   1:  PR[GP1:91,1] = PR[GP1:90,1] + -28.583;
   1:  PR[GP1:91,2] = PR[GP1:90,2] + 39.031;
   1:L PR[91] 10mm/sec CNT100;
   1:  PR[GP1:91,1] = PR[GP1:90,1] + -29.750;
   1:  PR[GP1:91,2] = PR[GP1:90,2] + 38.604;
   1:L PR[91] 10mm/sec CNT100;
   1:  PR[GP1:91,1] = PR[GP1:90,1] + -40.400;
   1:  PR[GP1:91,2] = PR[GP1:90,2] + 33.947;
   1:L PR[91] 10mm/sec CNT100;
   1:  PR[GP1:91,1] = PR[GP1:90,1] + -41.704;
   1:  PR[GP1:91,2] = PR[GP1:90,2] + 33.125;
   1:L PR[91] 10mm/sec CNT100;
   1:  PR[GP1:91,1] = PR[GP1:90,1] + -42.919;
   1:  PR[GP1:91,2] = PR[GP1:90,2] + 31.940;
   1:L PR[91] 10mm/sec CNT100;
   1:  PR[GP1:91,1] = PR[GP1:90,1] + -51.021;
   1:  PR[GP1:91,2] = PR[GP1:90,2] + 24.604;
   1:L PR[91] 10mm/sec CNT100;
   1:  PR[GP1:91,1] = PR[GP1:90,1] + -52.053;
   1:  PR[GP1:91,2] = PR[GP1:90,2] + 22.993;
   1:L PR[91] 10mm/sec CNT100;
   1:  PR[GP1:91,1] = PR[GP1:90,1] + -57.032;
   1:  PR[GP1:91,2] = PR[GP1:90,2] + 13.999;
   1:L PR[91] 10mm/sec CNT100;
   1:  PR[GP1:91,1] = PR[GP1:90,1] + -57.722;
   1:  PR[GP1:91,2] = PR[GP1:90,2] + 12.097;
   1:L PR[91] 10mm/sec CNT100;
   1:  PR[GP1:91,1] = PR[GP1:90,1] + -57.950;
   1:  PR[GP1:91,2] = PR[GP1:90,2] + 10.064;
   1:L PR[91] 10mm/sec CNT100;
   1:  PR[GP1:91,1] = PR[GP1:90,1] + -59.627;
   1:  PR[GP1:91,2] = PR[GP1:90,2] + 0.261;
   1:L PR[91] 10mm/sec CNT100;
   1:  PR[GP1:91,1] = PR[GP1:90,1] + -59.403;
   1:  PR[GP1:91,2] = PR[GP1:90,2] + -1.752;
   1:L PR[91] 10mm/sec CNT100;
   1:  PR[GP1:91,1] = PR[GP1:90,1] + -57.736;
   1:  PR[GP1:91,2] = PR[GP1:90,2] + -11.502;
   1:L PR[91] 10mm/sec CNT100;
   1:  PR[GP1:91,1] = PR[GP1:90,1] + -57.039;
   1:  PR[GP1:91,2] = PR[GP1:90,2] + -13.421;
   1:L PR[91] 10mm/sec CNT100;
   1:  PR[GP1:91,1] = PR[GP1:90,1] + -52.081;
   1:  PR[GP1:91,2] = PR[GP1:90,2] + -22.399;
   1:L PR[91] 10mm/sec CNT100;
   1:  PR[GP1:91,1] = PR[GP1:90,1] + -51.042;
   1:  PR[GP1:91,2] = PR[GP1:90,2] + -24.020;
   1:L PR[91] 10mm/sec CNT100;
   1:  PR[GP1:91,1] = PR[GP1:90,1] + -49.777;
   1:  PR[GP1:91,2] = PR[GP1:90,2] + -25.262;
   1:L PR[91] 10mm/sec CNT100;
   1:  PR[GP1:91,1] = PR[GP1:90,1] + -41.775;
   1:  PR[GP1:91,2] = PR[GP1:90,2] + -32.521;
   1:L PR[91] 10mm/sec CNT100;
   1:  PR[GP1:91,1] = PR[GP1:90,1] + -40.461;
   1:  PR[GP1:91,2] = PR[GP1:90,2] + -33.350;
   1:L PR[91] 10mm/sec CNT100;
   1:  PR[GP1:91,1] = PR[GP1:90,1] + -29.851;
   1:  PR[GP1:91,2] = PR[GP1:90,2] + -38.019;
   1:L PR[91] 10mm/sec CNT100;
   1:  PR[GP1:91,1] = PR[GP1:90,1] + -28.670;
   1:  PR[GP1:91,2] = PR[GP1:90,2] + -38.452;
   1:L PR[91] 10mm/sec CNT100;
   1:  PR[GP1:91,1] = PR[GP1:90,1] + -27.548;
   1:  PR[GP1:91,2] = PR[GP1:90,2] + -38.612;
   1:L PR[91] 10mm/sec CNT100;
   1:  PR[GP1:91,1] = PR[GP1:90,1] + -15.395;
   1:  PR[GP1:91,2] = PR[GP1:90,2] + -39.778;
   1:L PR[91] 10mm/sec CNT100;
   1:  PR[GP1:91,1] = PR[GP1:90,1] + -14.616;
   1:  PR[GP1:91,2] = PR[GP1:90,2] + -39.726;
   1:L PR[91] 10mm/sec CNT100;
   1:  PR[GP1:91,1] = PR[GP1:90,1] + -2.012;
   1:  PR[GP1:91,2] = PR[GP1:90,2] + -36.843;
   1:L PR[91] 10mm/sec CNT100;
   1:  PR[GP1:91,1] = PR[GP1:90,1] + -1.587;
   1:  PR[GP1:91,2] = PR[GP1:90,2] + -36.721;
   1:L PR[91] 10mm/sec CNT100;
   1:  PR[GP1:91,1] = PR[GP1:90,1] + -0.264;
   1:  PR[GP1:91,2] = PR[GP1:90,2] + -35.946;
   1:L PR[91] 10mm/sec CNT100;
   1:  PR[GP1:91,1] = PR[GP1:90,1] + 0.805;
   1:  PR[GP1:91,2] = PR[GP1:90,2] + -36.790;
   1:  PR[GP1:91,3] = PR[GP1:90,3] + 82.655;
   1:L PR[91] 10mm/sec CNT100;
   1:  PR[GP1:91,1] = PR[GP1:90,1] + 1.110;
   1:  PR[GP1:91,2] = PR[GP1:90,2] + -36.877;
   1:L PR[91] 10mm/sec CNT100;
   1:  PR[GP1:91,1] = PR[GP1:90,1] + 13.913;
   1:  PR[GP1:91,2] = PR[GP1:90,2] + -39.807;
   1:L PR[91] 10mm/sec CNT100;
   1:  PR[GP1:91,1] = PR[GP1:90,1] + 14.554;
   1:  PR[GP1:91,2] = PR[GP1:90,2] + -39.849;
   1:L PR[91] 10mm/sec CNT100;
   1:  PR[GP1:91,1] = PR[GP1:90,1] + 15.335;
   1:  PR[GP1:91,2] = PR[GP1:90,2] + -39.742;
   1:L PR[91] 10mm/sec CNT100;
   1:  PR[GP1:91,1] = PR[GP1:90,1] + 27.932;
   1:  PR[GP1:91,2] = PR[GP1:90,2] + -38.517;
   1:L PR[91] 10mm/sec CNT100;
   1:  PR[GP1:91,1] = PR[GP1:90,1] + 28.976;
   1:  PR[GP1:91,2] = PR[GP1:90,2] + -38.137;
   1:L PR[91] 10mm/sec CNT100;
   1:  PR[GP1:91,1] = PR[GP1:90,1] + 39.784;
   1:  PR[GP1:91,2] = PR[GP1:90,2] + -33.383;
   1:L PR[91] 10mm/sec CNT100;
   1:  PR[GP1:91,1] = PR[GP1:90,1] + 40.970;
   1:  PR[GP1:91,2] = PR[GP1:90,2] + -32.639;
   1:L PR[91] 10mm/sec CNT100;
   1:  PR[GP1:91,1] = PR[GP1:90,1] + 42.083;
   1:  PR[GP1:91,2] = PR[GP1:90,2] + -31.555;
   1:L PR[91] 10mm/sec CNT100;
   1:  PR[GP1:91,1] = PR[GP1:90,1] + 50.319;
   1:  PR[GP1:91,2] = PR[GP1:90,2] + -24.063;
   1:L PR[91] 10mm/sec CNT100;
   1:  PR[GP1:91,1] = PR[GP1:90,1] + 51.288;
   1:  PR[GP1:91,2] = PR[GP1:90,2] + -22.560;
   1:L PR[91] 10mm/sec CNT100;
   1:  PR[GP1:91,1] = PR[GP1:90,1] + 56.354;
   1:  PR[GP1:91,2] = PR[GP1:90,2] + -13.404;
   1:L PR[91] 10mm/sec CNT100;
   1:  PR[GP1:91,1] = PR[GP1:90,1] + 56.995;
   1:  PR[GP1:91,2] = PR[GP1:90,2] + -11.659;
   1:L PR[91] 10mm/sec CNT100;
   1:  PR[GP1:91,1] = PR[GP1:90,1] + 57.216;
   1:  PR[GP1:91,2] = PR[GP1:90,2] + -9.715;
   1:L PR[91] 10mm/sec CNT100;
   1:  PR[GP1:91,1] = PR[GP1:90,1] + 58.924;
   1:  PR[GP1:91,2] = PR[GP1:90,2] + 0.296;
   1:L PR[91] 10mm/sec CNT100;
   1:  PR[GP1:91,1] = PR[GP1:90,1] + 58.706;
   1:  PR[GP1:91,2] = PR[GP1:90,2] + 2.224;
   1:L PR[91] 10mm/sec CNT100;
   1:  PR[GP1:91,1] = PR[GP1:90,1] + 56.994;
   1:  PR[GP1:91,2] = PR[GP1:90,2] + 12.222;
   1:L PR[91] 10mm/sec CNT100;
   1:  PR[GP1:91,1] = PR[GP1:90,1] + 56.346;
   1:  PR[GP1:91,2] = PR[GP1:90,2] + 13.982;
   1:L PR[91] 10mm/sec CNT100;
   1:  PR[GP1:91,1] = PR[GP1:90,1] + 51.259;
   1:  PR[GP1:91,2] = PR[GP1:90,2] + 23.154;
   1:L PR[91] 10mm/sec CNT100;
   1:  PR[GP1:91,1] = PR[GP1:90,1] + 50.284;
   1:  PR[GP1:91,2] = PR[GP1:90,2] + 24.667;
   1:L PR[91] 10mm/sec CNT100;
   1:  PR[GP1:91,1] = PR[GP1:90,1] + 49.110;
   1:  PR[GP1:91,2] = PR[GP1:90,2] + 25.817;
   1:L PR[91] 10mm/sec CNT100;
   1:  PR[GP1:91,1] = PR[GP1:90,1] + 40.917;
   1:  PR[GP1:91,2] = PR[GP1:90,2] + 33.232;
   1:L PR[91] 10mm/sec CNT100;
   1:  PR[GP1:91,1] = PR[GP1:90,1] + 39.723;
   1:  PR[GP1:91,2] = PR[GP1:90,2] + 33.981;
   1:L PR[91] 10mm/sec CNT100;
   1:  PR[GP1:91,1] = PR[GP1:90,1] + 28.873;
   1:  PR[GP1:91,2] = PR[GP1:90,2] + 38.722;
   1:L PR[91] 10mm/sec CNT100;
   1:  PR[GP1:91,1] = PR[GP1:90,1] + 27.818;
   1:  PR[GP1:91,2] = PR[GP1:90,2] + 39.107;
   1:L PR[91] 10mm/sec CNT100;
   1:  PR[GP1:91,1] = PR[GP1:90,1] + 26.822;
   1:  PR[GP1:91,2] = PR[GP1:90,2] + 39.248;
   1:L PR[91] 10mm/sec CNT100;
   1:  PR[GP1:91,1] = PR[GP1:90,1] + 14.428;
   1:  PR[GP1:91,2] = PR[GP1:90,2] + 40.400;
   1:L PR[91] 10mm/sec CNT100;
   1:  PR[GP1:91,1] = PR[GP1:90,1] + 13.778;
   1:  PR[GP1:91,2] = PR[GP1:90,2] + 40.356;
   1:L PR[91] 10mm/sec CNT100;
   1:  PR[GP1:91,1] = PR[GP1:90,1] + 0.766;
   1:  PR[GP1:91,2] = PR[GP1:90,2] + 37.283;
   1:L PR[91] 10mm/sec CNT100;
   1:  PR[GP1:91,1] = PR[GP1:90,1] + 0.557;
   1:  PR[GP1:91,2] = PR[GP1:90,2] + 37.223;
   1:L PR[91] 10mm/sec CNT100;
   1:  PR[GP1:91,1] = PR[GP1:90,1] + -0.262;
   1:  PR[GP1:91,2] = PR[GP1:90,2] + 36.794;
   1:L PR[91] 10mm/sec CNT100;
   1:  PR[GP1:91,1] = PR[GP1:90,1] + -1.079;
   1:  PR[GP1:91,2] = PR[GP1:90,2] + 37.223;
   1:L PR[91] 10mm/sec CNT100;
   1:  PR[GP1:91,1] = PR[GP1:90,1] + -1.288;
   1:  PR[GP1:91,2] = PR[GP1:90,2] + 37.283;
   1:L PR[91] 10mm/sec CNT100;
   1:  PR[GP1:91,1] = PR[GP1:90,1] + -14.303;
   1:  PR[GP1:91,2] = PR[GP1:90,2] + 40.356;
   1:L PR[91] 10mm/sec CNT100;
   1:  PR[GP1:91,1] = PR[GP1:90,1] + -14.942;
   1:  PR[GP1:91,2] = PR[GP1:90,2] + 40.398;
   1:L PR[91] 10mm/sec CNT100;
   1:  PR[GP1:91,1] = PR[GP1:90,1] + -15.723;
   1:  PR[GP1:91,2] = PR[GP1:90,2] + 40.290;
   1:L PR[91] 10mm/sec CNT100;
   1:  PR[GP1:91,1] = PR[GP1:90,1] + -28.363;
   1:  PR[GP1:91,2] = PR[GP1:90,2] + 39.102;
   1:L PR[91] 10mm/sec CNT100;
   1:  PR[GP1:91,1] = PR[GP1:90,1] + -29.403;
   1:  PR[GP1:91,2] = PR[GP1:90,2] + 38.721;
   1:L PR[91] 10mm/sec CNT100;
   1:  PR[GP1:91,1] = PR[GP1:90,1] + -40.254;
   1:  PR[GP1:91,2] = PR[GP1:90,2] + 33.977;
   1:L PR[91] 10mm/sec CNT100;
   1:  PR[GP1:91,1] = PR[GP1:90,1] + -41.446;
   1:  PR[GP1:91,2] = PR[GP1:90,2] + 33.225;
   1:L PR[91] 10mm/sec CNT100;
   1:  PR[GP1:91,1] = PR[GP1:90,1] + -42.561;
   1:  PR[GP1:91,2] = PR[GP1:90,2] + 32.136;
   1:L PR[91] 10mm/sec CNT100;
   1:  PR[GP1:91,1] = PR[GP1:90,1] + -50.832;
   1:  PR[GP1:91,2] = PR[GP1:90,2] + 24.648;
   1:L PR[91] 10mm/sec CNT100;
   1:  PR[GP1:91,1] = PR[GP1:90,1] + -51.790;
   1:  PR[GP1:91,2] = PR[GP1:90,2] + 23.152;
   1:L PR[91] 10mm/sec CNT100;
   1:  PR[GP1:91,1] = PR[GP1:90,1] + -56.877;
   1:  PR[GP1:91,2] = PR[GP1:90,2] + 13.963;
   1:L PR[91] 10mm/sec CNT100;
   1:  PR[GP1:91,1] = PR[GP1:90,1] + -57.522;
   1:  PR[GP1:91,2] = PR[GP1:90,2] + 12.187;
   1:L PR[91] 10mm/sec CNT100;
   1:  PR[GP1:91,1] = PR[GP1:90,1] + -57.735;
   1:  PR[GP1:91,2] = PR[GP1:90,2] + 10.284;
   1:L PR[91] 10mm/sec CNT100;
   1:  PR[GP1:91,1] = PR[GP1:90,1] + -59.450;
   1:  PR[GP1:91,2] = PR[GP1:90,2] + 0.261;
   1:L PR[91] 10mm/sec CNT100;
   1:  PR[GP1:91,1] = PR[GP1:90,1] + -59.240;
   1:  PR[GP1:91,2] = PR[GP1:90,2] + -1.624;
   1:L PR[91] 10mm/sec CNT100;
   1:  PR[GP1:91,1] = PR[GP1:90,1] + -57.535;
   1:  PR[GP1:91,2] = PR[GP1:90,2] + -11.591;
   1:L PR[91] 10mm/sec CNT100;
   1:  PR[GP1:91,1] = PR[GP1:90,1] + -56.885;
   1:  PR[GP1:91,2] = PR[GP1:90,2] + -13.384;
   1:L PR[91] 10mm/sec CNT100;
   1:  PR[GP1:91,1] = PR[GP1:90,1] + -51.819;
   1:  PR[GP1:91,2] = PR[GP1:90,2] + -22.557;
   1:L PR[91] 10mm/sec CNT100;
   1:  PR[GP1:91,1] = PR[GP1:90,1] + -50.854;
   1:  PR[GP1:91,2] = PR[GP1:90,2] + -24.063;
   1:L PR[91] 10mm/sec CNT100;
   1:  PR[GP1:91,1] = PR[GP1:90,1] + -49.679;
   1:  PR[GP1:91,2] = PR[GP1:90,2] + -25.217;
   1:L PR[91] 10mm/sec CNT100;
   1:  PR[GP1:91,1] = PR[GP1:90,1] + -41.518;
   1:  PR[GP1:91,2] = PR[GP1:90,2] + -32.620;
   1:L PR[91] 10mm/sec CNT100;
   1:  PR[GP1:91,1] = PR[GP1:90,1] + -40.315;
   1:  PR[GP1:91,2] = PR[GP1:90,2] + -33.379;
   1:L PR[91] 10mm/sec CNT100;
   1:  PR[GP1:91,1] = PR[GP1:90,1] + -29.506;
   1:  PR[GP1:91,2] = PR[GP1:90,2] + -38.135;
   1:L PR[91] 10mm/sec CNT100;
   1:  PR[GP1:91,1] = PR[GP1:90,1] + -28.451;
   1:  PR[GP1:91,2] = PR[GP1:90,2] + -38.522;
   1:L PR[91] 10mm/sec CNT100;
   1:  PR[GP1:91,1] = PR[GP1:90,1] + -27.450;
   1:  PR[GP1:91,2] = PR[GP1:90,2] + -38.664;
   1:L PR[91] 10mm/sec CNT100;
   1:  PR[GP1:91,1] = PR[GP1:90,1] + -15.095;
   1:  PR[GP1:91,2] = PR[GP1:90,2] + -39.850;
   1:L PR[91] 10mm/sec CNT100;
   1:  PR[GP1:91,1] = PR[GP1:90,1] + -14.439;
   1:  PR[GP1:91,2] = PR[GP1:90,2] + -39.806;
   1:L PR[91] 10mm/sec CNT100;
   1:  PR[GP1:91,1] = PR[GP1:90,1] + -1.637;
   1:  PR[GP1:91,2] = PR[GP1:90,2] + -36.877;
   1:L PR[91] 10mm/sec CNT100;
   1:  PR[GP1:91,1] = PR[GP1:90,1] + -1.332;
   1:  PR[GP1:91,2] = PR[GP1:90,2] + -36.790;
   1:L PR[91] 10mm/sec CNT100;
   1:  PR[GP1:91,1] = PR[GP1:90,1] + -0.264;
   1:  PR[GP1:91,2] = PR[GP1:90,2] + -36.164;
   1:L PR[91] 10mm/sec CNT100;
   1:  PR[GP1:91,1] = PR[GP1:90,1] + 0.550;
   1:  PR[GP1:91,2] = PR[GP1:90,2] + -36.859;
   1:  PR[GP1:91,3] = PR[GP1:90,3] + 83.265;
   1:L PR[91] 10mm/sec CNT100;
   1:  PR[GP1:91,1] = PR[GP1:90,1] + 0.735;
   1:  PR[GP1:91,2] = PR[GP1:90,2] + -36.912;
   1:L PR[91] 10mm/sec CNT100;
   1:  PR[GP1:91,1] = PR[GP1:90,1] + 13.736;
   1:  PR[GP1:91,2] = PR[GP1:90,2] + -39.887;
   1:L PR[91] 10mm/sec CNT100;
   1:  PR[GP1:91,1] = PR[GP1:90,1] + 14.254;
   1:  PR[GP1:91,2] = PR[GP1:90,2] + -39.921;
   1:L PR[91] 10mm/sec CNT100;
   1:  PR[GP1:91,1] = PR[GP1:90,1] + 14.899;
   1:  PR[GP1:91,2] = PR[GP1:90,2] + -39.832;
   1:L PR[91] 10mm/sec CNT100;
   1:  PR[GP1:91,1] = PR[GP1:90,1] + 27.715;
   1:  PR[GP1:91,2] = PR[GP1:90,2] + -38.587;
   1:L PR[91] 10mm/sec CNT100;
   1:  PR[GP1:91,1] = PR[GP1:90,1] + 28.632;
   1:  PR[GP1:91,2] = PR[GP1:90,2] + -38.252;
   1:L PR[91] 10mm/sec CNT100;
   1:  PR[GP1:91,1] = PR[GP1:90,1] + 39.639;
   1:  PR[GP1:91,2] = PR[GP1:90,2] + -33.412;
   1:L PR[91] 10mm/sec CNT100;
   1:  PR[GP1:91,1] = PR[GP1:90,1] + 40.715;
   1:  PR[GP1:91,2] = PR[GP1:90,2] + -32.737;
   1:L PR[91] 10mm/sec CNT100;
   1:  PR[GP1:91,1] = PR[GP1:90,1] + 41.728;
   1:  PR[GP1:91,2] = PR[GP1:90,2] + -31.749;
   1:L PR[91] 10mm/sec CNT100;
   1:  PR[GP1:91,1] = PR[GP1:90,1] + 50.132;
   1:  PR[GP1:91,2] = PR[GP1:90,2] + -24.105;
   1:L PR[91] 10mm/sec CNT100;
   1:  PR[GP1:91,1] = PR[GP1:90,1] + 51.027;
   1:  PR[GP1:91,2] = PR[GP1:90,2] + -22.717;
   1:L PR[91] 10mm/sec CNT100;
   1:  PR[GP1:91,1] = PR[GP1:90,1] + 56.200;
   1:  PR[GP1:91,2] = PR[GP1:90,2] + -13.367;
   1:L PR[91] 10mm/sec CNT100;
   1:  PR[GP1:91,1] = PR[GP1:90,1] + 56.796;
   1:  PR[GP1:91,2] = PR[GP1:90,2] + -11.746;
   1:L PR[91] 10mm/sec CNT100;
   1:  PR[GP1:91,1] = PR[GP1:90,1] + 57.002;
   1:  PR[GP1:91,2] = PR[GP1:90,2] + -9.935;
   1:L PR[91] 10mm/sec CNT100;
   1:  PR[GP1:91,1] = PR[GP1:90,1] + 58.747;
   1:  PR[GP1:91,2] = PR[GP1:90,2] + 0.296;
   1:L PR[91] 10mm/sec CNT100;
   1:  PR[GP1:91,1] = PR[GP1:90,1] + 58.543;
   1:  PR[GP1:91,2] = PR[GP1:90,2] + 2.093;
   1:L PR[91] 10mm/sec CNT100;
   1:  PR[GP1:91,1] = PR[GP1:90,1] + 56.794;
   1:  PR[GP1:91,2] = PR[GP1:90,2] + 12.309;
   1:L PR[91] 10mm/sec CNT100;
   1:  PR[GP1:91,1] = PR[GP1:90,1] + 56.192;
   1:  PR[GP1:91,2] = PR[GP1:90,2] + 13.946;
   1:L PR[91] 10mm/sec CNT100;
   1:  PR[GP1:91,1] = PR[GP1:90,1] + 50.997;
   1:  PR[GP1:91,2] = PR[GP1:90,2] + 23.313;
   1:L PR[91] 10mm/sec CNT100;
   1:  PR[GP1:91,1] = PR[GP1:90,1] + 50.096;
   1:  PR[GP1:91,2] = PR[GP1:90,2] + 24.710;
   1:L PR[91] 10mm/sec CNT100;
   1:  PR[GP1:91,1] = PR[GP1:90,1] + 49.013;
   1:  PR[GP1:91,2] = PR[GP1:90,2] + 25.771;
   1:L PR[91] 10mm/sec CNT100;
   1:  PR[GP1:91,1] = PR[GP1:90,1] + 40.660;
   1:  PR[GP1:91,2] = PR[GP1:90,2] + 33.330;
   1:L PR[91] 10mm/sec CNT100;
   1:  PR[GP1:91,1] = PR[GP1:90,1] + 39.577;
   1:  PR[GP1:91,2] = PR[GP1:90,2] + 34.010;
   1:L PR[91] 10mm/sec CNT100;
   1:  PR[GP1:91,1] = PR[GP1:90,1] + 28.527;
   1:  PR[GP1:91,2] = PR[GP1:90,2] + 38.838;
   1:L PR[91] 10mm/sec CNT100;
   1:  PR[GP1:91,1] = PR[GP1:90,1] + 27.599;
   1:  PR[GP1:91,2] = PR[GP1:90,2] + 39.177;
   1:L PR[91] 10mm/sec CNT100;
   1:  PR[GP1:91,1] = PR[GP1:90,1] + 26.723;
   1:  PR[GP1:91,2] = PR[GP1:90,2] + 39.301;
   1:L PR[91] 10mm/sec CNT100;
   1:  PR[GP1:91,1] = PR[GP1:90,1] + 14.126;
   1:  PR[GP1:91,2] = PR[GP1:90,2] + 40.471;
   1:L PR[91] 10mm/sec CNT100;
   1:  PR[GP1:91,1] = PR[GP1:90,1] + 13.599;
   1:  PR[GP1:91,2] = PR[GP1:90,2] + 40.436;
   1:L PR[91] 10mm/sec CNT100;
   1:  PR[GP1:91,1] = PR[GP1:90,1] + 0.385;
   1:  PR[GP1:91,2] = PR[GP1:90,2] + 37.316;
   1:L PR[91] 10mm/sec CNT100;
   1:  PR[GP1:91,1] = PR[GP1:90,1] + 0.299;
   1:  PR[GP1:91,2] = PR[GP1:90,2] + 37.291;
   1:L PR[91] 10mm/sec CNT100;
   1:  PR[GP1:91,1] = PR[GP1:90,1] + -0.262;
   1:  PR[GP1:91,2] = PR[GP1:90,2] + 36.997;
   1:L PR[91] 10mm/sec CNT100;
   1:  PR[GP1:91,1] = PR[GP1:90,1] + -0.821;
   1:  PR[GP1:91,2] = PR[GP1:90,2] + 37.291;
   1:L PR[91] 10mm/sec CNT100;
   1:  PR[GP1:91,1] = PR[GP1:90,1] + -0.907;
   1:  PR[GP1:91,2] = PR[GP1:90,2] + 37.316;
   1:L PR[91] 10mm/sec CNT100;
   1:  PR[GP1:91,1] = PR[GP1:90,1] + -14.124;
   1:  PR[GP1:91,2] = PR[GP1:90,2] + 40.436;
   1:L PR[91] 10mm/sec CNT100;
   1:  PR[GP1:91,1] = PR[GP1:90,1] + -14.639;
   1:  PR[GP1:91,2] = PR[GP1:90,2] + 40.470;
   1:L PR[91] 10mm/sec CNT100;
   1:  PR[GP1:91,1] = PR[GP1:90,1] + -15.284;
   1:  PR[GP1:91,2] = PR[GP1:90,2] + 40.381;
   1:L PR[91] 10mm/sec CNT100;
   1:  PR[GP1:91,1] = PR[GP1:90,1] + -28.143;
   1:  PR[GP1:91,2] = PR[GP1:90,2] + 39.172;
   1:L PR[91] 10mm/sec CNT100;
   1:  PR[GP1:91,1] = PR[GP1:90,1] + -29.057;
   1:  PR[GP1:91,2] = PR[GP1:90,2] + 38.837;
   1:L PR[91] 10mm/sec CNT100;
   1:  PR[GP1:91,1] = PR[GP1:90,1] + -40.107;
   1:  PR[GP1:91,2] = PR[GP1:90,2] + 34.006;
   1:L PR[91] 10mm/sec CNT100;
   1:  PR[GP1:91,1] = PR[GP1:90,1] + -41.188;
   1:  PR[GP1:91,2] = PR[GP1:90,2] + 33.324;
   1:L PR[91] 10mm/sec CNT100;
   1:  PR[GP1:91,1] = PR[GP1:90,1] + -42.203;
   1:  PR[GP1:91,2] = PR[GP1:90,2] + 32.333;
   1:L PR[91] 10mm/sec CNT100;
   1:  PR[GP1:91,1] = PR[GP1:90,1] + -50.643;
   1:  PR[GP1:91,2] = PR[GP1:90,2] + 24.691;
   1:L PR[91] 10mm/sec CNT100;
   1:  PR[GP1:91,1] = PR[GP1:90,1] + -51.527;
   1:  PR[GP1:91,2] = PR[GP1:90,2] + 23.311;
   1:L PR[91] 10mm/sec CNT100;
   1:  PR[GP1:91,1] = PR[GP1:90,1] + -56.723;
   1:  PR[GP1:91,2] = PR[GP1:90,2] + 13.927;
   1:L PR[91] 10mm/sec CNT100;
   1:  PR[GP1:91,1] = PR[GP1:90,1] + -57.322;
   1:  PR[GP1:91,2] = PR[GP1:90,2] + 12.277;
   1:L PR[91] 10mm/sec CNT100;
   1:  PR[GP1:91,1] = PR[GP1:90,1] + -57.520;
   1:  PR[GP1:91,2] = PR[GP1:90,2] + 10.504;
   1:L PR[91] 10mm/sec CNT100;
   1:  PR[GP1:91,1] = PR[GP1:90,1] + -59.273;
   1:  PR[GP1:91,2] = PR[GP1:90,2] + 0.261;
   1:L PR[91] 10mm/sec CNT100;
   1:  PR[GP1:91,1] = PR[GP1:90,1] + -59.077;
   1:  PR[GP1:91,2] = PR[GP1:90,2] + -1.496;
   1:L PR[91] 10mm/sec CNT100;
   1:  PR[GP1:91,1] = PR[GP1:90,1] + -57.335;
   1:  PR[GP1:91,2] = PR[GP1:90,2] + -11.681;
   1:L PR[91] 10mm/sec CNT100;
   1:  PR[GP1:91,1] = PR[GP1:90,1] + -56.730;
   1:  PR[GP1:91,2] = PR[GP1:90,2] + -13.348;
   1:L PR[91] 10mm/sec CNT100;
   1:  PR[GP1:91,1] = PR[GP1:90,1] + -51.557;
   1:  PR[GP1:91,2] = PR[GP1:90,2] + -22.716;
   1:L PR[91] 10mm/sec CNT100;
   1:  PR[GP1:91,1] = PR[GP1:90,1] + -50.666;
   1:  PR[GP1:91,2] = PR[GP1:90,2] + -24.106;
   1:L PR[91] 10mm/sec CNT100;
   1:  PR[GP1:91,1] = PR[GP1:90,1] + -49.581;
   1:  PR[GP1:91,2] = PR[GP1:90,2] + -25.171;
   1:L PR[91] 10mm/sec CNT100;
   1:  PR[GP1:91,1] = PR[GP1:90,1] + -41.262;
   1:  PR[GP1:91,2] = PR[GP1:90,2] + -32.718;
   1:L PR[91] 10mm/sec CNT100;
   1:  PR[GP1:91,1] = PR[GP1:90,1] + -40.169;
   1:  PR[GP1:91,2] = PR[GP1:90,2] + -33.407;
   1:L PR[91] 10mm/sec CNT100;
   1:  PR[GP1:91,1] = PR[GP1:90,1] + -29.162;
   1:  PR[GP1:91,2] = PR[GP1:90,2] + -38.251;
   1:L PR[91] 10mm/sec CNT100;
   1:  PR[GP1:91,1] = PR[GP1:90,1] + -28.233;
   1:  PR[GP1:91,2] = PR[GP1:90,2] + -38.592;
   1:L PR[91] 10mm/sec CNT100;
   1:  PR[GP1:91,1] = PR[GP1:90,1] + -27.352;
   1:  PR[GP1:91,2] = PR[GP1:90,2] + -38.717;
   1:L PR[91] 10mm/sec CNT100;
   1:  PR[GP1:91,1] = PR[GP1:90,1] + -14.795;
   1:  PR[GP1:91,2] = PR[GP1:90,2] + -39.922;
   1:L PR[91] 10mm/sec CNT100;
   1:  PR[GP1:91,1] = PR[GP1:90,1] + -14.262;
   1:  PR[GP1:91,2] = PR[GP1:90,2] + -39.887;
   1:L PR[91] 10mm/sec CNT100;
   1:  PR[GP1:91,1] = PR[GP1:90,1] + -1.261;
   1:  PR[GP1:91,2] = PR[GP1:90,2] + -36.912;
   1:L PR[91] 10mm/sec CNT100;
   1:  PR[GP1:91,1] = PR[GP1:90,1] + -1.077;
   1:  PR[GP1:91,2] = PR[GP1:90,2] + -36.859;
   1:L PR[91] 10mm/sec CNT100;
   1:  PR[GP1:91,1] = PR[GP1:90,1] + -0.264;
   1:  PR[GP1:91,2] = PR[GP1:90,2] + -36.383;
   1:L PR[91] 10mm/sec CNT100;
   1:  PR[GP1:91,1] = PR[GP1:90,1] + 0.296;
   1:  PR[GP1:91,2] = PR[GP1:90,2] + -36.929;
   1:  PR[GP1:91,3] = PR[GP1:90,3] + 83.875;
   1:L PR[91] 10mm/sec CNT100;
   1:  PR[GP1:91,1] = PR[GP1:90,1] + 0.360;
   1:  PR[GP1:91,2] = PR[GP1:90,2] + -36.947;
   1:L PR[91] 10mm/sec CNT100;
   1:  PR[GP1:91,1] = PR[GP1:90,1] + 13.559;
   1:  PR[GP1:91,2] = PR[GP1:90,2] + -39.967;
   1:L PR[91] 10mm/sec CNT100;
   1:  PR[GP1:91,1] = PR[GP1:90,1] + 13.954;
   1:  PR[GP1:91,2] = PR[GP1:90,2] + -39.993;
   1:L PR[91] 10mm/sec CNT100;
   1:  PR[GP1:91,1] = PR[GP1:90,1] + 14.463;
   1:  PR[GP1:91,2] = PR[GP1:90,2] + -39.923;
   1:L PR[91] 10mm/sec CNT100;
   1:  PR[GP1:91,1] = PR[GP1:90,1] + 27.497;
   1:  PR[GP1:91,2] = PR[GP1:90,2] + -38.657;
   1:L PR[91] 10mm/sec CNT100;
   1:  PR[GP1:91,1] = PR[GP1:90,1] + 28.287;
   1:  PR[GP1:91,2] = PR[GP1:90,2] + -38.368;
   1:L PR[91] 10mm/sec CNT100;
   1:  PR[GP1:91,1] = PR[GP1:90,1] + 39.494;
   1:  PR[GP1:91,2] = PR[GP1:90,2] + -33.440;
   1:L PR[91] 10mm/sec CNT100;
   1:  PR[GP1:91,1] = PR[GP1:90,1] + 40.459;
   1:  PR[GP1:91,2] = PR[GP1:90,2] + -32.834;
   1:L PR[91] 10mm/sec CNT100;
   1:  PR[GP1:91,1] = PR[GP1:90,1] + 41.373;
   1:  PR[GP1:91,2] = PR[GP1:90,2] + -31.944;
   1:L PR[91] 10mm/sec CNT100;
   1:  PR[GP1:91,1] = PR[GP1:90,1] + 49.945;
   1:  PR[GP1:91,2] = PR[GP1:90,2] + -24.146;
   1:L PR[91] 10mm/sec CNT100;
   1:  PR[GP1:91,1] = PR[GP1:90,1] + 50.765;
   1:  PR[GP1:91,2] = PR[GP1:90,2] + -22.875;
   1:L PR[91] 10mm/sec CNT100;
   1:  PR[GP1:91,1] = PR[GP1:90,1] + 56.045;
   1:  PR[GP1:91,2] = PR[GP1:90,2] + -13.330;
   1:L PR[91] 10mm/sec CNT100;
   1:  PR[GP1:91,1] = PR[GP1:90,1] + 56.596;
   1:  PR[GP1:91,2] = PR[GP1:90,2] + -11.833;
   1:L PR[91] 10mm/sec CNT100;
   1:  PR[GP1:91,1] = PR[GP1:90,1] + 56.787;
   1:  PR[GP1:91,2] = PR[GP1:90,2] + -10.155;
   1:L PR[91] 10mm/sec CNT100;
   1:  PR[GP1:91,1] = PR[GP1:90,1] + 58.569;
   1:  PR[GP1:91,2] = PR[GP1:90,2] + 0.296;
   1:L PR[91] 10mm/sec CNT100;
   1:  PR[GP1:91,1] = PR[GP1:90,1] + 58.381;
   1:  PR[GP1:91,2] = PR[GP1:90,2] + 1.962;
   1:L PR[91] 10mm/sec CNT100;
   1:  PR[GP1:91,1] = PR[GP1:90,1] + 56.594;
   1:  PR[GP1:91,2] = PR[GP1:90,2] + 12.396;
   1:L PR[91] 10mm/sec CNT100;
   1:  PR[GP1:91,1] = PR[GP1:90,1] + 56.038;
   1:  PR[GP1:91,2] = PR[GP1:90,2] + 13.909;
   1:L PR[91] 10mm/sec CNT100;
   1:  PR[GP1:91,1] = PR[GP1:90,1] + 50.735;
   1:  PR[GP1:91,2] = PR[GP1:90,2] + 23.471;
   1:L PR[91] 10mm/sec CNT100;
   1:  PR[GP1:91,1] = PR[GP1:90,1] + 49.909;
   1:  PR[GP1:91,2] = PR[GP1:90,2] + 24.752;
   1:L PR[91] 10mm/sec CNT100;
   1:  PR[GP1:91,1] = PR[GP1:90,1] + 48.916;
   1:  PR[GP1:91,2] = PR[GP1:90,2] + 25.725;
   1:L PR[91] 10mm/sec CNT100;
   1:  PR[GP1:91,1] = PR[GP1:90,1] + 40.404;
   1:  PR[GP1:91,2] = PR[GP1:90,2] + 33.428;
   1:L PR[91] 10mm/sec CNT100;
   1:  PR[GP1:91,1] = PR[GP1:90,1] + 39.430;
   1:  PR[GP1:91,2] = PR[GP1:90,2] + 34.039;
   1:L PR[91] 10mm/sec CNT100;
   1:  PR[GP1:91,1] = PR[GP1:90,1] + 28.181;
   1:  PR[GP1:91,2] = PR[GP1:90,2] + 38.954;
   1:L PR[91] 10mm/sec CNT100;
   1:  PR[GP1:91,1] = PR[GP1:90,1] + 27.379;
   1:  PR[GP1:91,2] = PR[GP1:90,2] + 39.247;
   1:L PR[91] 10mm/sec CNT100;
   1:  PR[GP1:91,1] = PR[GP1:90,1] + 26.624;
   1:  PR[GP1:91,2] = PR[GP1:90,2] + 39.354;
   1:L PR[91] 10mm/sec CNT100;
   1:  PR[GP1:91,1] = PR[GP1:90,1] + 13.824;
   1:  PR[GP1:91,2] = PR[GP1:90,2] + 40.543;
   1:L PR[91] 10mm/sec CNT100;
   1:  PR[GP1:91,1] = PR[GP1:90,1] + 13.420;
   1:  PR[GP1:91,2] = PR[GP1:90,2] + 40.516;
   1:L PR[91] 10mm/sec CNT100;
   1:  PR[GP1:91,1] = PR[GP1:90,1] + 0.046;
   1:  PR[GP1:91,2] = PR[GP1:90,2] + 37.358;
   1:L PR[91] 10mm/sec CNT100;
   1:  PR[GP1:91,1] = PR[GP1:90,1] + -0.261;
   1:  PR[GP1:91,2] = PR[GP1:90,2] + 37.220;
   1:L PR[91] 10mm/sec CNT100;
   1:  PR[GP1:91,1] = PR[GP1:90,1] + -0.568;
   1:  PR[GP1:91,2] = PR[GP1:90,2] + 37.358;
   1:L PR[91] 10mm/sec CNT100;
   1:  PR[GP1:91,1] = PR[GP1:90,1] + -13.945;
   1:  PR[GP1:91,2] = PR[GP1:90,2] + 40.516;
   1:L PR[91] 10mm/sec CNT100;
   1:  PR[GP1:91,1] = PR[GP1:90,1] + -14.337;
   1:  PR[GP1:91,2] = PR[GP1:90,2] + 40.542;
   1:L PR[91] 10mm/sec CNT100;
   1:  PR[GP1:91,1] = PR[GP1:90,1] + -14.845;
   1:  PR[GP1:91,2] = PR[GP1:90,2] + 40.471;
   1:L PR[91] 10mm/sec CNT100;
   1:  PR[GP1:91,1] = PR[GP1:90,1] + -27.923;
   1:  PR[GP1:91,2] = PR[GP1:90,2] + 39.242;
   1:L PR[91] 10mm/sec CNT100;
   1:  PR[GP1:91,1] = PR[GP1:90,1] + -28.710;
   1:  PR[GP1:91,2] = PR[GP1:90,2] + 38.954;
   1:L PR[91] 10mm/sec CNT100;
   1:  PR[GP1:91,1] = PR[GP1:90,1] + -39.960;
   1:  PR[GP1:91,2] = PR[GP1:90,2] + 34.035;
   1:L PR[91] 10mm/sec CNT100;
   1:  PR[GP1:91,1] = PR[GP1:90,1] + -40.930;
   1:  PR[GP1:91,2] = PR[GP1:90,2] + 33.423;
   1:L PR[91] 10mm/sec CNT100;
   1:  PR[GP1:91,1] = PR[GP1:90,1] + -41.846;
   1:  PR[GP1:91,2] = PR[GP1:90,2] + 32.530;
   1:L PR[91] 10mm/sec CNT100;
   1:  PR[GP1:91,1] = PR[GP1:90,1] + -50.455;
   1:  PR[GP1:91,2] = PR[GP1:90,2] + 24.735;
   1:L PR[91] 10mm/sec CNT100;
   1:  PR[GP1:91,1] = PR[GP1:90,1] + -51.265;
   1:  PR[GP1:91,2] = PR[GP1:90,2] + 23.471;
   1:L PR[91] 10mm/sec CNT100;
   1:  PR[GP1:91,1] = PR[GP1:90,1] + -56.568;
   1:  PR[GP1:91,2] = PR[GP1:90,2] + 13.891;
   1:L PR[91] 10mm/sec CNT100;
   1:  PR[GP1:91,1] = PR[GP1:90,1] + -57.121;
   1:  PR[GP1:91,2] = PR[GP1:90,2] + 12.366;
   1:L PR[91] 10mm/sec CNT100;
   1:  PR[GP1:91,1] = PR[GP1:90,1] + -57.305;
   1:  PR[GP1:91,2] = PR[GP1:90,2] + 10.724;
   1:L PR[91] 10mm/sec CNT100;
   1:  PR[GP1:91,1] = PR[GP1:90,1] + -59.096;
   1:  PR[GP1:91,2] = PR[GP1:90,2] + 0.261;
   1:L PR[91] 10mm/sec CNT100;
   1:  PR[GP1:91,1] = PR[GP1:90,1] + -58.914;
   1:  PR[GP1:91,2] = PR[GP1:90,2] + -1.368;
   1:L PR[91] 10mm/sec CNT100;
   1:  PR[GP1:91,1] = PR[GP1:90,1] + -57.135;
   1:  PR[GP1:91,2] = PR[GP1:90,2] + -11.770;
   1:L PR[91] 10mm/sec CNT100;
   1:  PR[GP1:91,1] = PR[GP1:90,1] + -56.576;
   1:  PR[GP1:91,2] = PR[GP1:90,2] + -13.312;
   1:L PR[91] 10mm/sec CNT100;
   1:  PR[GP1:91,1] = PR[GP1:90,1] + -51.295;
   1:  PR[GP1:91,2] = PR[GP1:90,2] + -22.874;
   1:L PR[91] 10mm/sec CNT100;
   1:  PR[GP1:91,1] = PR[GP1:90,1] + -50.478;
   1:  PR[GP1:91,2] = PR[GP1:90,2] + -24.149;
   1:L PR[91] 10mm/sec CNT100;
   1:  PR[GP1:91,1] = PR[GP1:90,1] + -49.483;
   1:  PR[GP1:91,2] = PR[GP1:90,2] + -25.125;
   1:L PR[91] 10mm/sec CNT100;
   1:  PR[GP1:91,1] = PR[GP1:90,1] + -41.005;
   1:  PR[GP1:91,2] = PR[GP1:90,2] + -32.817;
   1:L PR[91] 10mm/sec CNT100;
   1:  PR[GP1:91,1] = PR[GP1:90,1] + -40.024;
   1:  PR[GP1:91,2] = PR[GP1:90,2] + -33.436;
   1:L PR[91] 10mm/sec CNT100;
   1:  PR[GP1:91,1] = PR[GP1:90,1] + -28.817;
   1:  PR[GP1:91,2] = PR[GP1:90,2] + -38.368;
   1:L PR[91] 10mm/sec CNT100;
   1:  PR[GP1:91,1] = PR[GP1:90,1] + -28.015;
   1:  PR[GP1:91,2] = PR[GP1:90,2] + -38.661;
   1:L PR[91] 10mm/sec CNT100;
   1:  PR[GP1:91,1] = PR[GP1:90,1] + -27.255;
   1:  PR[GP1:91,2] = PR[GP1:90,2] + -38.770;
   1:L PR[91] 10mm/sec CNT100;
   1:  PR[GP1:91,1] = PR[GP1:90,1] + -14.494;
   1:  PR[GP1:91,2] = PR[GP1:90,2] + -39.994;
   1:L PR[91] 10mm/sec CNT100;
   1:  PR[GP1:91,1] = PR[GP1:90,1] + -14.085;
   1:  PR[GP1:91,2] = PR[GP1:90,2] + -39.967;
   1:L PR[91] 10mm/sec CNT100;
   1:  PR[GP1:91,1] = PR[GP1:90,1] + -0.886;
   1:  PR[GP1:91,2] = PR[GP1:90,2] + -36.947;
   1:L PR[91] 10mm/sec CNT100;
   1:  PR[GP1:91,1] = PR[GP1:90,1] + -0.822;
   1:  PR[GP1:91,2] = PR[GP1:90,2] + -36.929;
   1:L PR[91] 10mm/sec CNT100;
   1:  PR[GP1:91,1] = PR[GP1:90,1] + -0.264;
   1:  PR[GP1:91,2] = PR[GP1:90,2] + -36.601;
   1:L PR[91] 10mm/sec CNT100;
   1:  PR[GP1:91,1] = PR[GP1:90,1] + 0.036;
   1:  PR[GP1:91,2] = PR[GP1:90,2] + -36.994;
   1:  PR[GP1:91,3] = PR[GP1:90,3] + 84.485;
   1:L PR[91] 10mm/sec CNT100;
   1:  PR[GP1:91,1] = PR[GP1:90,1] + 13.382;
   1:  PR[GP1:91,2] = PR[GP1:90,2] + -40.047;
   1:L PR[91] 10mm/sec CNT100;
   1:  PR[GP1:91,1] = PR[GP1:90,1] + 13.654;
   1:  PR[GP1:91,2] = PR[GP1:90,2] + -40.065;
   1:L PR[91] 10mm/sec CNT100;
   1:  PR[GP1:91,1] = PR[GP1:90,1] + 14.027;
   1:  PR[GP1:91,2] = PR[GP1:90,2] + -40.014;
   1:L PR[91] 10mm/sec CNT100;
   1:  PR[GP1:91,1] = PR[GP1:90,1] + 27.280;
   1:  PR[GP1:91,2] = PR[GP1:90,2] + -38.726;
   1:L PR[91] 10mm/sec CNT100;
   1:  PR[GP1:91,1] = PR[GP1:90,1] + 27.943;
   1:  PR[GP1:91,2] = PR[GP1:90,2] + -38.484;
   1:L PR[91] 10mm/sec CNT100;
   1:  PR[GP1:91,1] = PR[GP1:90,1] + 39.348;
   1:  PR[GP1:91,2] = PR[GP1:90,2] + -33.468;
   1:L PR[91] 10mm/sec CNT100;
   1:  PR[GP1:91,1] = PR[GP1:90,1] + 40.203;
   1:  PR[GP1:91,2] = PR[GP1:90,2] + -32.932;
   1:L PR[91] 10mm/sec CNT100;
   1:  PR[GP1:91,1] = PR[GP1:90,1] + 41.018;
   1:  PR[GP1:91,2] = PR[GP1:90,2] + -32.138;
   1:L PR[91] 10mm/sec CNT100;
   1:  PR[GP1:91,1] = PR[GP1:90,1] + 49.758;
   1:  PR[GP1:91,2] = PR[GP1:90,2] + -24.188;
   1:L PR[91] 10mm/sec CNT100;
   1:  PR[GP1:91,1] = PR[GP1:90,1] + 50.503;
   1:  PR[GP1:91,2] = PR[GP1:90,2] + -23.033;
   1:L PR[91] 10mm/sec CNT100;
   1:  PR[GP1:91,1] = PR[GP1:90,1] + 55.891;
   1:  PR[GP1:91,2] = PR[GP1:90,2] + -13.293;
   1:L PR[91] 10mm/sec CNT100;
   1:  PR[GP1:91,1] = PR[GP1:90,1] + 56.397;
   1:  PR[GP1:91,2] = PR[GP1:90,2] + -11.919;
   1:L PR[91] 10mm/sec CNT100;
   1:  PR[GP1:91,1] = PR[GP1:90,1] + 56.572;
   1:  PR[GP1:91,2] = PR[GP1:90,2] + -10.374;
   1:L PR[91] 10mm/sec CNT100;
   1:  PR[GP1:91,1] = PR[GP1:90,1] + 58.392;
   1:  PR[GP1:91,2] = PR[GP1:90,2] + 0.296;
   1:L PR[91] 10mm/sec CNT100;
   1:  PR[GP1:91,1] = PR[GP1:90,1] + 58.218;
   1:  PR[GP1:91,2] = PR[GP1:90,2] + 1.832;
   1:L PR[91] 10mm/sec CNT100;
   1:  PR[GP1:91,1] = PR[GP1:90,1] + 56.395;
   1:  PR[GP1:91,2] = PR[GP1:90,2] + 12.483;
   1:L PR[91] 10mm/sec CNT100;
   1:  PR[GP1:91,1] = PR[GP1:90,1] + 55.884;
   1:  PR[GP1:91,2] = PR[GP1:90,2] + 13.873;
   1:L PR[91] 10mm/sec CNT100;
   1:  PR[GP1:91,1] = PR[GP1:90,1] + 50.472;
   1:  PR[GP1:91,2] = PR[GP1:90,2] + 23.630;
   1:L PR[91] 10mm/sec CNT100;
   1:  PR[GP1:91,1] = PR[GP1:90,1] + 49.722;
   1:  PR[GP1:91,2] = PR[GP1:90,2] + 24.794;
   1:L PR[91] 10mm/sec CNT100;
   1:  PR[GP1:91,1] = PR[GP1:90,1] + 48.818;
   1:  PR[GP1:91,2] = PR[GP1:90,2] + 25.679;
   1:L PR[91] 10mm/sec CNT100;
   1:  PR[GP1:91,1] = PR[GP1:90,1] + 40.147;
   1:  PR[GP1:91,2] = PR[GP1:90,2] + 33.527;
   1:L PR[91] 10mm/sec CNT100;
   1:  PR[GP1:91,1] = PR[GP1:90,1] + 39.284;
   1:  PR[GP1:91,2] = PR[GP1:90,2] + 34.068;
   1:L PR[91] 10mm/sec CNT100;
   1:  PR[GP1:91,1] = PR[GP1:90,1] + 27.835;
   1:  PR[GP1:91,2] = PR[GP1:90,2] + 39.070;
   1:L PR[91] 10mm/sec CNT100;
   1:  PR[GP1:91,1] = PR[GP1:90,1] + 27.160;
   1:  PR[GP1:91,2] = PR[GP1:90,2] + 39.317;
   1:L PR[91] 10mm/sec CNT100;
   1:  PR[GP1:91,1] = PR[GP1:90,1] + 26.525;
   1:  PR[GP1:91,2] = PR[GP1:90,2] + 39.407;
   1:L PR[91] 10mm/sec CNT100;
   1:  PR[GP1:91,1] = PR[GP1:90,1] + 13.521;
   1:  PR[GP1:91,2] = PR[GP1:90,2] + 40.615;
   1:L PR[91] 10mm/sec CNT100;
   1:  PR[GP1:91,1] = PR[GP1:90,1] + 13.241;
   1:  PR[GP1:91,2] = PR[GP1:90,2] + 40.596;
   1:L PR[91] 10mm/sec CNT100;
   1:  PR[GP1:91,1] = PR[GP1:90,1] + 2.271;
   1:  PR[GP1:91,2] = PR[GP1:90,2] + 38.006;
   1:L PR[91] 10mm/sec CNT100;
   1:  PR[GP1:91,1] = PR[GP1:90,1] + -0.261;
   1:  PR[GP1:91,2] = PR[GP1:90,2] + 37.453;
   1:L PR[91] 10mm/sec CNT100;
   1:  PR[GP1:91,1] = PR[GP1:90,1] + -2.794;
   1:  PR[GP1:91,2] = PR[GP1:90,2] + 38.006;
   1:L PR[91] 10mm/sec CNT100;
   1:  PR[GP1:91,1] = PR[GP1:90,1] + -13.767;
   1:  PR[GP1:91,2] = PR[GP1:90,2] + 40.596;
   1:L PR[91] 10mm/sec CNT100;
   1:  PR[GP1:91,1] = PR[GP1:90,1] + -14.034;
   1:  PR[GP1:91,2] = PR[GP1:90,2] + 40.614;
   1:L PR[91] 10mm/sec CNT100;
   1:  PR[GP1:91,1] = PR[GP1:90,1] + -14.405;
   1:  PR[GP1:91,2] = PR[GP1:90,2] + 40.562;
   1:L PR[91] 10mm/sec CNT100;
   1:  PR[GP1:91,1] = PR[GP1:90,1] + -27.703;
   1:  PR[GP1:91,2] = PR[GP1:90,2] + 39.312;
   1:L PR[91] 10mm/sec CNT100;
   1:  PR[GP1:91,1] = PR[GP1:90,1] + -28.364;
   1:  PR[GP1:91,2] = PR[GP1:90,2] + 39.070;
   1:L PR[91] 10mm/sec CNT100;
   1:  PR[GP1:91,1] = PR[GP1:90,1] + -39.813;
   1:  PR[GP1:91,2] = PR[GP1:90,2] + 34.064;
   1:L PR[91] 10mm/sec CNT100;
   1:  PR[GP1:91,1] = PR[GP1:90,1] + -40.672;
   1:  PR[GP1:91,2] = PR[GP1:90,2] + 33.523;
   1:L PR[91] 10mm/sec CNT100;
   1:  PR[GP1:91,1] = PR[GP1:90,1] + -41.488;
   1:  PR[GP1:91,2] = PR[GP1:90,2] + 32.726;
   1:L PR[91] 10mm/sec CNT100;
   1:  PR[GP1:91,1] = PR[GP1:90,1] + -50.266;
   1:  PR[GP1:91,2] = PR[GP1:90,2] + 24.779;
   1:L PR[91] 10mm/sec CNT100;
   1:  PR[GP1:91,1] = PR[GP1:90,1] + -51.002;
   1:  PR[GP1:91,2] = PR[GP1:90,2] + 23.630;
   1:L PR[91] 10mm/sec CNT100;
   1:  PR[GP1:91,1] = PR[GP1:90,1] + -56.413;
   1:  PR[GP1:91,2] = PR[GP1:90,2] + 13.855;
   1:L PR[91] 10mm/sec CNT100;
   1:  PR[GP1:91,1] = PR[GP1:90,1] + -56.921;
   1:  PR[GP1:91,2] = PR[GP1:90,2] + 12.456;
   1:L PR[91] 10mm/sec CNT100;
   1:  PR[GP1:91,1] = PR[GP1:90,1] + -57.091;
   1:  PR[GP1:91,2] = PR[GP1:90,2] + 10.944;
   1:L PR[91] 10mm/sec CNT100;
   1:  PR[GP1:91,1] = PR[GP1:90,1] + -58.919;
   1:  PR[GP1:91,2] = PR[GP1:90,2] + 0.261;
   1:L PR[91] 10mm/sec CNT100;
   1:  PR[GP1:91,1] = PR[GP1:90,1] + -58.751;
   1:  PR[GP1:91,2] = PR[GP1:90,2] + -1.240;
   1:L PR[91] 10mm/sec CNT100;
   1:  PR[GP1:91,1] = PR[GP1:90,1] + -56.935;
   1:  PR[GP1:91,2] = PR[GP1:90,2] + -11.859;
   1:L PR[91] 10mm/sec CNT100;
   1:  PR[GP1:91,1] = PR[GP1:90,1] + -56.421;
   1:  PR[GP1:91,2] = PR[GP1:90,2] + -13.275;
   1:L PR[91] 10mm/sec CNT100;
   1:  PR[GP1:91,1] = PR[GP1:90,1] + -51.033;
   1:  PR[GP1:91,2] = PR[GP1:90,2] + -23.032;
   1:L PR[91] 10mm/sec CNT100;
   1:  PR[GP1:91,1] = PR[GP1:90,1] + -50.290;
   1:  PR[GP1:91,2] = PR[GP1:90,2] + -24.192;
   1:L PR[91] 10mm/sec CNT100;
   1:  PR[GP1:91,1] = PR[GP1:90,1] + -49.385;
   1:  PR[GP1:91,2] = PR[GP1:90,2] + -25.080;
   1:L PR[91] 10mm/sec CNT100;
   1:  PR[GP1:91,1] = PR[GP1:90,1] + -40.748;
   1:  PR[GP1:91,2] = PR[GP1:90,2] + -32.915;
   1:L PR[91] 10mm/sec CNT100;
   1:  PR[GP1:91,1] = PR[GP1:90,1] + -39.878;
   1:  PR[GP1:91,2] = PR[GP1:90,2] + -33.464;
   1:L PR[91] 10mm/sec CNT100;
   1:  PR[GP1:91,1] = PR[GP1:90,1] + -28.472;
   1:  PR[GP1:91,2] = PR[GP1:90,2] + -38.484;
   1:L PR[91] 10mm/sec CNT100;
   1:  PR[GP1:91,1] = PR[GP1:90,1] + -27.797;
   1:  PR[GP1:91,2] = PR[GP1:90,2] + -38.731;
   1:L PR[91] 10mm/sec CNT100;
   1:  PR[GP1:91,1] = PR[GP1:90,1] + -27.157;
   1:  PR[GP1:91,2] = PR[GP1:90,2] + -38.822;
   1:L PR[91] 10mm/sec CNT100;
   1:  PR[GP1:91,1] = PR[GP1:90,1] + -14.194;
   1:  PR[GP1:91,2] = PR[GP1:90,2] + -40.066;
   1:L PR[91] 10mm/sec CNT100;
   1:  PR[GP1:91,1] = PR[GP1:90,1] + -13.909;
   1:  PR[GP1:91,2] = PR[GP1:90,2] + -40.047;
   1:L PR[91] 10mm/sec CNT100;
   1:  PR[GP1:91,1] = PR[GP1:90,1] + -0.562;
   1:  PR[GP1:91,2] = PR[GP1:90,2] + -36.994;
   1:L PR[91] 10mm/sec CNT100;
   1:  PR[GP1:91,1] = PR[GP1:90,1] + -0.263;
   1:  PR[GP1:91,2] = PR[GP1:90,2] + -36.847;
   1:L PR[91] 10mm/sec CNT100;
   1:  PR[GP1:91,1] = PR[GP1:90,1] + 3.266;
   1:  PR[GP1:91,2] = PR[GP1:90,2] + -37.853;
   1:  PR[GP1:91,3] = PR[GP1:90,3] + 85.095;
   1:L PR[91] 10mm/sec CNT100;
   1:  PR[GP1:91,1] = PR[GP1:90,1] + 13.206;
   1:  PR[GP1:91,2] = PR[GP1:90,2] + -40.128;
   1:L PR[91] 10mm/sec CNT100;
   1:  PR[GP1:91,1] = PR[GP1:90,1] + 13.354;
   1:  PR[GP1:91,2] = PR[GP1:90,2] + -40.137;
   1:L PR[91] 10mm/sec CNT100;
   1:  PR[GP1:91,1] = PR[GP1:90,1] + 13.591;
   1:  PR[GP1:91,2] = PR[GP1:90,2] + -40.105;
   1:L PR[91] 10mm/sec CNT100;
   1:  PR[GP1:91,1] = PR[GP1:90,1] + 27.062;
   1:  PR[GP1:91,2] = PR[GP1:90,2] + -38.796;
   1:L PR[91] 10mm/sec CNT100;
   1:  PR[GP1:91,1] = PR[GP1:90,1] + 27.599;
   1:  PR[GP1:91,2] = PR[GP1:90,2] + -38.600;
   1:L PR[91] 10mm/sec CNT100;
   1:  PR[GP1:91,1] = PR[GP1:90,1] + 39.203;
   1:  PR[GP1:91,2] = PR[GP1:90,2] + -33.497;
   1:L PR[91] 10mm/sec CNT100;
   1:  PR[GP1:91,1] = PR[GP1:90,1] + 39.948;
   1:  PR[GP1:91,2] = PR[GP1:90,2] + -33.029;
   1:L PR[91] 10mm/sec CNT100;
   1:  PR[GP1:91,1] = PR[GP1:90,1] + 40.663;
   1:  PR[GP1:91,2] = PR[GP1:90,2] + -32.333;
   1:L PR[91] 10mm/sec CNT100;
   1:  PR[GP1:91,1] = PR[GP1:90,1] + 49.571;
   1:  PR[GP1:91,2] = PR[GP1:90,2] + -24.229;
   1:L PR[91] 10mm/sec CNT100;
   1:  PR[GP1:91,1] = PR[GP1:90,1] + 50.241;
   1:  PR[GP1:91,2] = PR[GP1:90,2] + -23.190;
   1:L PR[91] 10mm/sec CNT100;
   1:  PR[GP1:91,1] = PR[GP1:90,1] + 55.737;
   1:  PR[GP1:91,2] = PR[GP1:90,2] + -13.257;
   1:L PR[91] 10mm/sec CNT100;
   1:  PR[GP1:91,1] = PR[GP1:90,1] + 56.197;
   1:  PR[GP1:91,2] = PR[GP1:90,2] + -12.006;
   1:L PR[91] 10mm/sec CNT100;
   1:  PR[GP1:91,1] = PR[GP1:90,1] + 56.357;
   1:  PR[GP1:91,2] = PR[GP1:90,2] + -10.594;
   1:L PR[91] 10mm/sec CNT100;
   1:  PR[GP1:91,1] = PR[GP1:90,1] + 58.215;
   1:  PR[GP1:91,2] = PR[GP1:90,2] + 0.296;
   1:L PR[91] 10mm/sec CNT100;
   1:  PR[GP1:91,1] = PR[GP1:90,1] + 58.056;
   1:  PR[GP1:91,2] = PR[GP1:90,2] + 1.701;
   1:L PR[91] 10mm/sec CNT100;
   1:  PR[GP1:91,1] = PR[GP1:90,1] + 56.195;
   1:  PR[GP1:91,2] = PR[GP1:90,2] + 12.570;
   1:L PR[91] 10mm/sec CNT100;
   1:  PR[GP1:91,1] = PR[GP1:90,1] + 55.729;
   1:  PR[GP1:91,2] = PR[GP1:90,2] + 13.837;
   1:L PR[91] 10mm/sec CNT100;
   1:  PR[GP1:91,1] = PR[GP1:90,1] + 50.210;
   1:  PR[GP1:91,2] = PR[GP1:90,2] + 23.788;
   1:L PR[91] 10mm/sec CNT100;
   1:  PR[GP1:91,1] = PR[GP1:90,1] + 49.534;
   1:  PR[GP1:91,2] = PR[GP1:90,2] + 24.836;
   1:L PR[91] 10mm/sec CNT100;
   1:  PR[GP1:91,1] = PR[GP1:90,1] + 48.721;
   1:  PR[GP1:91,2] = PR[GP1:90,2] + 25.633;
   1:L PR[91] 10mm/sec CNT100;
   1:  PR[GP1:91,1] = PR[GP1:90,1] + 39.890;
   1:  PR[GP1:91,2] = PR[GP1:90,2] + 33.625;
   1:L PR[91] 10mm/sec CNT100;
   1:  PR[GP1:91,1] = PR[GP1:90,1] + 39.138;
   1:  PR[GP1:91,2] = PR[GP1:90,2] + 34.097;
   1:L PR[91] 10mm/sec CNT100;
   1:  PR[GP1:91,1] = PR[GP1:90,1] + 27.489;
   1:  PR[GP1:91,2] = PR[GP1:90,2] + 39.187;
   1:L PR[91] 10mm/sec CNT100;
   1:  PR[GP1:91,1] = PR[GP1:90,1] + 26.941;
   1:  PR[GP1:91,2] = PR[GP1:90,2] + 39.387;
   1:L PR[91] 10mm/sec CNT100;
   1:  PR[GP1:91,1] = PR[GP1:90,1] + 26.426;
   1:  PR[GP1:91,2] = PR[GP1:90,2] + 39.460;
   1:L PR[91] 10mm/sec CNT100;
   1:  PR[GP1:91,1] = PR[GP1:90,1] + 13.219;
   1:  PR[GP1:91,2] = PR[GP1:90,2] + 40.687;
   1:L PR[91] 10mm/sec CNT100;
   1:  PR[GP1:91,1] = PR[GP1:90,1] + 13.062;
   1:  PR[GP1:91,2] = PR[GP1:90,2] + 40.677;
   1:L PR[91] 10mm/sec CNT100;
   1:  PR[GP1:91,1] = PR[GP1:90,1] + 5.691;
   1:  PR[GP1:91,2] = PR[GP1:90,2] + 38.935;
   1:L PR[91] 10mm/sec CNT100;
   1:  PR[GP1:91,1] = PR[GP1:90,1] + -0.261;
   1:  PR[GP1:91,2] = PR[GP1:90,2] + 37.637;
   1:L PR[91] 10mm/sec CNT100;
   1:  PR[GP1:91,1] = PR[GP1:90,1] + -6.214;
   1:  PR[GP1:91,2] = PR[GP1:90,2] + 38.935;
   1:L PR[91] 10mm/sec CNT100;
   1:  PR[GP1:91,1] = PR[GP1:90,1] + -13.588;
   1:  PR[GP1:91,2] = PR[GP1:90,2] + 40.676;
   1:L PR[91] 10mm/sec CNT100;
   1:  PR[GP1:91,1] = PR[GP1:90,1] + -13.732;
   1:  PR[GP1:91,2] = PR[GP1:90,2] + 40.686;
   1:L PR[91] 10mm/sec CNT100;
   1:  PR[GP1:91,1] = PR[GP1:90,1] + -13.966;
   1:  PR[GP1:91,2] = PR[GP1:90,2] + 40.653;
   1:L PR[91] 10mm/sec CNT100;
   1:  PR[GP1:91,1] = PR[GP1:90,1] + -27.483;
   1:  PR[GP1:91,2] = PR[GP1:90,2] + 39.382;
   1:L PR[91] 10mm/sec CNT100;
   1:  PR[GP1:91,1] = PR[GP1:90,1] + -28.017;
   1:  PR[GP1:91,2] = PR[GP1:90,2] + 39.187;
   1:L PR[91] 10mm/sec CNT100;
   1:  PR[GP1:91,1] = PR[GP1:90,1] + -39.666;
   1:  PR[GP1:91,2] = PR[GP1:90,2] + 34.093;
   1:L PR[91] 10mm/sec CNT100;
   1:  PR[GP1:91,1] = PR[GP1:90,1] + -40.414;
   1:  PR[GP1:91,2] = PR[GP1:90,2] + 33.622;
   1:L PR[91] 10mm/sec CNT100;
   1:  PR[GP1:91,1] = PR[GP1:90,1] + -41.130;
   1:  PR[GP1:91,2] = PR[GP1:90,2] + 32.923;
   1:L PR[91] 10mm/sec CNT100;
   1:  PR[GP1:91,1] = PR[GP1:90,1] + -50.077;
   1:  PR[GP1:91,2] = PR[GP1:90,2] + 24.822;
   1:L PR[91] 10mm/sec CNT100;
   1:  PR[GP1:91,1] = PR[GP1:90,1] + -50.739;
   1:  PR[GP1:91,2] = PR[GP1:90,2] + 23.789;
   1:L PR[91] 10mm/sec CNT100;
   1:  PR[GP1:91,1] = PR[GP1:90,1] + -56.259;
   1:  PR[GP1:91,2] = PR[GP1:90,2] + 13.819;
   1:L PR[91] 10mm/sec CNT100;
   1:  PR[GP1:91,1] = PR[GP1:90,1] + -56.721;
   1:  PR[GP1:91,2] = PR[GP1:90,2] + 12.546;
   1:L PR[91] 10mm/sec CNT100;
   1:  PR[GP1:91,1] = PR[GP1:90,1] + -56.876;
   1:  PR[GP1:91,2] = PR[GP1:90,2] + 11.164;
   1:L PR[91] 10mm/sec CNT100;
   1:  PR[GP1:91,1] = PR[GP1:90,1] + -58.741;
   1:  PR[GP1:91,2] = PR[GP1:90,2] + 0.261;
   1:L PR[91] 10mm/sec CNT100;
   1:  PR[GP1:91,1] = PR[GP1:90,1] + -58.588;
   1:  PR[GP1:91,2] = PR[GP1:90,2] + -1.112;
   1:L PR[91] 10mm/sec CNT100;
   1:  PR[GP1:91,1] = PR[GP1:90,1] + -56.735;
   1:  PR[GP1:91,2] = PR[GP1:90,2] + -11.949;
   1:L PR[91] 10mm/sec CNT100;
   1:  PR[GP1:91,1] = PR[GP1:90,1] + -56.267;
   1:  PR[GP1:91,2] = PR[GP1:90,2] + -13.239;
   1:L PR[91] 10mm/sec CNT100;
   1:  PR[GP1:91,1] = PR[GP1:90,1] + -50.771;
   1:  PR[GP1:91,2] = PR[GP1:90,2] + -23.191;
   1:L PR[91] 10mm/sec CNT100;
   1:  PR[GP1:91,1] = PR[GP1:90,1] + -50.102;
   1:  PR[GP1:91,2] = PR[GP1:90,2] + -24.235;
   1:L PR[91] 10mm/sec CNT100;
   1:  PR[GP1:91,1] = PR[GP1:90,1] + -49.287;
   1:  PR[GP1:91,2] = PR[GP1:90,2] + -25.034;
   1:L PR[91] 10mm/sec CNT100;
   1:  PR[GP1:91,1] = PR[GP1:90,1] + -40.491;
   1:  PR[GP1:91,2] = PR[GP1:90,2] + -33.014;
   1:L PR[91] 10mm/sec CNT100;
   1:  PR[GP1:91,1] = PR[GP1:90,1] + -39.732;
   1:  PR[GP1:91,2] = PR[GP1:90,2] + -33.493;
   1:L PR[91] 10mm/sec CNT100;
   1:  PR[GP1:91,1] = PR[GP1:90,1] + -28.128;
   1:  PR[GP1:91,2] = PR[GP1:90,2] + -38.600;
   1:L PR[91] 10mm/sec CNT100;
   1:  PR[GP1:91,1] = PR[GP1:90,1] + -27.579;
   1:  PR[GP1:91,2] = PR[GP1:90,2] + -38.801;
   1:L PR[91] 10mm/sec CNT100;
   1:  PR[GP1:91,1] = PR[GP1:90,1] + -27.059;
   1:  PR[GP1:91,2] = PR[GP1:90,2] + -38.875;
   1:L PR[91] 10mm/sec CNT100;
   1:  PR[GP1:91,1] = PR[GP1:90,1] + -13.894;
   1:  PR[GP1:91,2] = PR[GP1:90,2] + -40.138;
   1:L PR[91] 10mm/sec CNT100;
   1:  PR[GP1:91,1] = PR[GP1:90,1] + -13.732;
   1:  PR[GP1:91,2] = PR[GP1:90,2] + -40.127;
   1:L PR[91] 10mm/sec CNT100;
   1:  PR[GP1:91,1] = PR[GP1:90,1] + -3.793;
   1:  PR[GP1:91,2] = PR[GP1:90,2] + -37.853;
   1:L PR[91] 10mm/sec CNT100;
   1:  PR[GP1:91,1] = PR[GP1:90,1] + -0.263;
   1:  PR[GP1:91,2] = PR[GP1:90,2] + -37.100;
   1:L PR[91] 10mm/sec CNT100;
   1:  PR[GP1:91,1] = PR[GP1:90,1] + 7.861;
   1:  PR[GP1:91,2] = PR[GP1:90,2] + -39.025;
   1:  PR[GP1:91,3] = PR[GP1:90,3] + 85.705;
   1:L PR[91] 10mm/sec CNT100;
   1:  PR[GP1:91,1] = PR[GP1:90,1] + 13.029;
   1:  PR[GP1:91,2] = PR[GP1:90,2] + -40.208;
   1:L PR[91] 10mm/sec CNT100;
   1:  PR[GP1:91,1] = PR[GP1:90,1] + 13.067;
   1:  PR[GP1:91,2] = PR[GP1:90,2] + -40.210;
   1:L PR[91] 10mm/sec CNT100;
   1:  PR[GP1:91,1] = PR[GP1:90,1] + 26.844;
   1:  PR[GP1:91,2] = PR[GP1:90,2] + -38.865;
   1:L PR[91] 10mm/sec CNT100;
   1:  PR[GP1:91,1] = PR[GP1:90,1] + 27.255;
   1:  PR[GP1:91,2] = PR[GP1:90,2] + -38.715;
   1:L PR[91] 10mm/sec CNT100;
   1:  PR[GP1:91,1] = PR[GP1:90,1] + 39.058;
   1:  PR[GP1:91,2] = PR[GP1:90,2] + -33.525;
   1:L PR[91] 10mm/sec CNT100;
   1:  PR[GP1:91,1] = PR[GP1:90,1] + 39.692;
   1:  PR[GP1:91,2] = PR[GP1:90,2] + -33.127;
   1:L PR[91] 10mm/sec CNT100;
   1:  PR[GP1:91,1] = PR[GP1:90,1] + 40.308;
   1:  PR[GP1:91,2] = PR[GP1:90,2] + -32.527;
   1:L PR[91] 10mm/sec CNT100;
   1:  PR[GP1:91,1] = PR[GP1:90,1] + 49.384;
   1:  PR[GP1:91,2] = PR[GP1:90,2] + -24.271;
   1:L PR[91] 10mm/sec CNT100;
   1:  PR[GP1:91,1] = PR[GP1:90,1] + 49.980;
   1:  PR[GP1:91,2] = PR[GP1:90,2] + -23.348;
   1:L PR[91] 10mm/sec CNT100;
   1:  PR[GP1:91,1] = PR[GP1:90,1] + 55.583;
   1:  PR[GP1:91,2] = PR[GP1:90,2] + -13.220;
   1:L PR[91] 10mm/sec CNT100;
   1:  PR[GP1:91,1] = PR[GP1:90,1] + 55.997;
   1:  PR[GP1:91,2] = PR[GP1:90,2] + -12.093;
   1:L PR[91] 10mm/sec CNT100;
   1:  PR[GP1:91,1] = PR[GP1:90,1] + 56.143;
   1:  PR[GP1:91,2] = PR[GP1:90,2] + -10.814;
   1:L PR[91] 10mm/sec CNT100;
   1:  PR[GP1:91,1] = PR[GP1:90,1] + 58.038;
   1:  PR[GP1:91,2] = PR[GP1:90,2] + 0.296;
   1:L PR[91] 10mm/sec CNT100;
   1:  PR[GP1:91,1] = PR[GP1:90,1] + 57.894;
   1:  PR[GP1:91,2] = PR[GP1:90,2] + 1.571;
   1:L PR[91] 10mm/sec CNT100;
   1:  PR[GP1:91,1] = PR[GP1:90,1] + 55.995;
   1:  PR[GP1:91,2] = PR[GP1:90,2] + 12.658;
   1:L PR[91] 10mm/sec CNT100;
   1:  PR[GP1:91,1] = PR[GP1:90,1] + 55.575;
   1:  PR[GP1:91,2] = PR[GP1:90,2] + 13.800;
   1:L PR[91] 10mm/sec CNT100;
   1:  PR[GP1:91,1] = PR[GP1:90,1] + 49.948;
   1:  PR[GP1:91,2] = PR[GP1:90,2] + 23.946;
   1:L PR[91] 10mm/sec CNT100;
   1:  PR[GP1:91,1] = PR[GP1:90,1] + 49.347;
   1:  PR[GP1:91,2] = PR[GP1:90,2] + 24.879;
   1:L PR[91] 10mm/sec CNT100;
   1:  PR[GP1:91,1] = PR[GP1:90,1] + 48.623;
   1:  PR[GP1:91,2] = PR[GP1:90,2] + 25.587;
   1:L PR[91] 10mm/sec CNT100;
   1:  PR[GP1:91,1] = PR[GP1:90,1] + 39.633;
   1:  PR[GP1:91,2] = PR[GP1:90,2] + 33.723;
   1:L PR[91] 10mm/sec CNT100;
   1:  PR[GP1:91,1] = PR[GP1:90,1] + 38.991;
   1:  PR[GP1:91,2] = PR[GP1:90,2] + 34.126;
   1:L PR[91] 10mm/sec CNT100;
   1:  PR[GP1:91,1] = PR[GP1:90,1] + 27.143;
   1:  PR[GP1:91,2] = PR[GP1:90,2] + 39.303;
   1:L PR[91] 10mm/sec CNT100;
   1:  PR[GP1:91,1] = PR[GP1:90,1] + 26.722;
   1:  PR[GP1:91,2] = PR[GP1:90,2] + 39.457;
   1:L PR[91] 10mm/sec CNT100;
   1:  PR[GP1:91,1] = PR[GP1:90,1] + 26.326;
   1:  PR[GP1:91,2] = PR[GP1:90,2] + 39.513;
   1:L PR[91] 10mm/sec CNT100;
   1:  PR[GP1:91,1] = PR[GP1:90,1] + 12.917;
   1:  PR[GP1:91,2] = PR[GP1:90,2] + 40.759;
   1:L PR[91] 10mm/sec CNT100;
   1:  PR[GP1:91,1] = PR[GP1:90,1] + 12.883;
   1:  PR[GP1:91,2] = PR[GP1:90,2] + 40.757;
   1:L PR[91] 10mm/sec CNT100;
   1:  PR[GP1:91,1] = PR[GP1:90,1] + 9.110;
   1:  PR[GP1:91,2] = PR[GP1:90,2] + 39.865;
   1:L PR[91] 10mm/sec CNT100;
   1:  PR[GP1:91,1] = PR[GP1:90,1] + -0.261;
   1:  PR[GP1:91,2] = PR[GP1:90,2] + 37.821;
   1:L PR[91] 10mm/sec CNT100;
   1:  PR[GP1:91,1] = PR[GP1:90,1] + -9.634;
   1:  PR[GP1:91,2] = PR[GP1:90,2] + 39.865;
   1:L PR[91] 10mm/sec CNT100;
   1:  PR[GP1:91,1] = PR[GP1:90,1] + -13.409;
   1:  PR[GP1:91,2] = PR[GP1:90,2] + 40.756;
   1:L PR[91] 10mm/sec CNT100;
   1:  PR[GP1:91,1] = PR[GP1:90,1] + -13.442;
   1:  PR[GP1:91,2] = PR[GP1:90,2] + 40.758;
   1:L PR[91] 10mm/sec CNT100;
   1:  PR[GP1:91,1] = PR[GP1:90,1] + -27.263;
   1:  PR[GP1:91,2] = PR[GP1:90,2] + 39.453;
   1:L PR[91] 10mm/sec CNT100;
   1:  PR[GP1:91,1] = PR[GP1:90,1] + -27.670;
   1:  PR[GP1:91,2] = PR[GP1:90,2] + 39.303;
   1:L PR[91] 10mm/sec CNT100;
   1:  PR[GP1:91,1] = PR[GP1:90,1] + -39.520;
   1:  PR[GP1:91,2] = PR[GP1:90,2] + 34.123;
   1:L PR[91] 10mm/sec CNT100;
   1:  PR[GP1:91,1] = PR[GP1:90,1] + -40.156;
   1:  PR[GP1:91,2] = PR[GP1:90,2] + 33.721;
   1:L PR[91] 10mm/sec CNT100;
   1:  PR[GP1:91,1] = PR[GP1:90,1] + -40.773;
   1:  PR[GP1:91,2] = PR[GP1:90,2] + 33.119;
   1:L PR[91] 10mm/sec CNT100;
   1:  PR[GP1:91,1] = PR[GP1:90,1] + -49.889;
   1:  PR[GP1:91,2] = PR[GP1:90,2] + 24.866;
   1:L PR[91] 10mm/sec CNT100;
   1:  PR[GP1:91,1] = PR[GP1:90,1] + -50.477;
   1:  PR[GP1:91,2] = PR[GP1:90,2] + 23.948;
   1:L PR[91] 10mm/sec CNT100;
   1:  PR[GP1:91,1] = PR[GP1:90,1] + -56.104;
   1:  PR[GP1:91,2] = PR[GP1:90,2] + 13.783;
   1:L PR[91] 10mm/sec CNT100;
   1:  PR[GP1:91,1] = PR[GP1:90,1] + -56.521;
   1:  PR[GP1:91,2] = PR[GP1:90,2] + 12.636;
   1:L PR[91] 10mm/sec CNT100;
   1:  PR[GP1:91,1] = PR[GP1:90,1] + -56.661;
   1:  PR[GP1:91,2] = PR[GP1:90,2] + 11.384;
   1:L PR[91] 10mm/sec CNT100;
   1:  PR[GP1:91,1] = PR[GP1:90,1] + -58.564;
   1:  PR[GP1:91,2] = PR[GP1:90,2] + 0.261;
   1:L PR[91] 10mm/sec CNT100;
   1:  PR[GP1:91,1] = PR[GP1:90,1] + -58.425;
   1:  PR[GP1:91,2] = PR[GP1:90,2] + -0.984;
   1:L PR[91] 10mm/sec CNT100;
   1:  PR[GP1:91,1] = PR[GP1:90,1] + -56.535;
   1:  PR[GP1:91,2] = PR[GP1:90,2] + -12.038;
   1:L PR[91] 10mm/sec CNT100;
   1:  PR[GP1:91,1] = PR[GP1:90,1] + -56.112;
   1:  PR[GP1:91,2] = PR[GP1:90,2] + -13.202;
   1:L PR[91] 10mm/sec CNT100;
   1:  PR[GP1:91,1] = PR[GP1:90,1] + -50.509;
   1:  PR[GP1:91,2] = PR[GP1:90,2] + -23.349;
   1:L PR[91] 10mm/sec CNT100;
   1:  PR[GP1:91,1] = PR[GP1:90,1] + -49.914;
   1:  PR[GP1:91,2] = PR[GP1:90,2] + -24.278;
   1:L PR[91] 10mm/sec CNT100;
   1:  PR[GP1:91,1] = PR[GP1:90,1] + -49.189;
   1:  PR[GP1:91,2] = PR[GP1:90,2] + -24.989;
   1:L PR[91] 10mm/sec CNT100;
   1:  PR[GP1:91,1] = PR[GP1:90,1] + -40.235;
   1:  PR[GP1:91,2] = PR[GP1:90,2] + -33.112;
   1:L PR[91] 10mm/sec CNT100;
   1:  PR[GP1:91,1] = PR[GP1:90,1] + -39.587;
   1:  PR[GP1:91,2] = PR[GP1:90,2] + -33.521;
   1:L PR[91] 10mm/sec CNT100;
   1:  PR[GP1:91,1] = PR[GP1:90,1] + -27.783;
   1:  PR[GP1:91,2] = PR[GP1:90,2] + -38.716;
   1:L PR[91] 10mm/sec CNT100;
   1:  PR[GP1:91,1] = PR[GP1:90,1] + -27.361;
   1:  PR[GP1:91,2] = PR[GP1:90,2] + -38.871;
   1:L PR[91] 10mm/sec CNT100;
   1:  PR[GP1:91,1] = PR[GP1:90,1] + -26.961;
   1:  PR[GP1:91,2] = PR[GP1:90,2] + -38.927;
   1:L PR[91] 10mm/sec CNT100;
   1:  PR[GP1:91,1] = PR[GP1:90,1] + -13.594;
   1:  PR[GP1:91,2] = PR[GP1:90,2] + -40.210;
   1:L PR[91] 10mm/sec CNT100;
   1:  PR[GP1:91,1] = PR[GP1:90,1] + -13.555;
   1:  PR[GP1:91,2] = PR[GP1:90,2] + -40.207;
   1:L PR[91] 10mm/sec CNT100;
   1:  PR[GP1:91,1] = PR[GP1:90,1] + -8.389;
   1:  PR[GP1:91,2] = PR[GP1:90,2] + -39.025;
   1:L PR[91] 10mm/sec CNT100;
   1:  PR[GP1:91,1] = PR[GP1:90,1] + -0.263;
   1:  PR[GP1:91,2] = PR[GP1:90,2] + -37.281;
   1:L PR[91] 10mm/sec CNT100;
   1:  PR[GP1:91,1] = PR[GP1:90,1] + 12.811;
   1:  PR[GP1:91,2] = PR[GP1:90,2] + -40.278;
   1:  PR[GP1:91,3] = PR[GP1:90,3] + 86.315;
   1:L PR[91] 10mm/sec CNT100;
   1:  PR[GP1:91,1] = PR[GP1:90,1] + 26.627;
   1:  PR[GP1:91,2] = PR[GP1:90,2] + -38.935;
   1:L PR[91] 10mm/sec CNT100;
   1:  PR[GP1:91,1] = PR[GP1:90,1] + 26.911;
   1:  PR[GP1:91,2] = PR[GP1:90,2] + -38.831;
   1:L PR[91] 10mm/sec CNT100;
   1:  PR[GP1:91,1] = PR[GP1:90,1] + 38.913;
   1:  PR[GP1:91,2] = PR[GP1:90,2] + -33.553;
   1:L PR[91] 10mm/sec CNT100;
   1:  PR[GP1:91,1] = PR[GP1:90,1] + 39.437;
   1:  PR[GP1:91,2] = PR[GP1:90,2] + -33.225;
   1:L PR[91] 10mm/sec CNT100;
   1:  PR[GP1:91,1] = PR[GP1:90,1] + 39.952;
   1:  PR[GP1:91,2] = PR[GP1:90,2] + -32.722;
   1:L PR[91] 10mm/sec CNT100;
   1:  PR[GP1:91,1] = PR[GP1:90,1] + 49.198;
   1:  PR[GP1:91,2] = PR[GP1:90,2] + -24.313;
   1:L PR[91] 10mm/sec CNT100;
   1:  PR[GP1:91,1] = PR[GP1:90,1] + 49.718;
   1:  PR[GP1:91,2] = PR[GP1:90,2] + -23.505;
   1:L PR[91] 10mm/sec CNT100;
   1:  PR[GP1:91,1] = PR[GP1:90,1] + 55.429;
   1:  PR[GP1:91,2] = PR[GP1:90,2] + -13.183;
   1:L PR[91] 10mm/sec CNT100;
   1:  PR[GP1:91,1] = PR[GP1:90,1] + 55.798;
   1:  PR[GP1:91,2] = PR[GP1:90,2] + -12.179;
   1:L PR[91] 10mm/sec CNT100;
   1:  PR[GP1:91,1] = PR[GP1:90,1] + 55.928;
   1:  PR[GP1:91,2] = PR[GP1:90,2] + -11.034;
   1:L PR[91] 10mm/sec CNT100;
   1:  PR[GP1:91,1] = PR[GP1:90,1] + 57.860;
   1:  PR[GP1:91,2] = PR[GP1:90,2] + 0.296;
   1:L PR[91] 10mm/sec CNT100;
   1:  PR[GP1:91,1] = PR[GP1:90,1] + 57.731;
   1:  PR[GP1:91,2] = PR[GP1:90,2] + 1.440;
   1:L PR[91] 10mm/sec CNT100;
   1:  PR[GP1:91,1] = PR[GP1:90,1] + 55.795;
   1:  PR[GP1:91,2] = PR[GP1:90,2] + 12.745;
   1:L PR[91] 10mm/sec CNT100;
   1:  PR[GP1:91,1] = PR[GP1:90,1] + 55.421;
   1:  PR[GP1:91,2] = PR[GP1:90,2] + 13.764;
   1:L PR[91] 10mm/sec CNT100;
   1:  PR[GP1:91,1] = PR[GP1:90,1] + 49.685;
   1:  PR[GP1:91,2] = PR[GP1:90,2] + 24.105;
   1:L PR[91] 10mm/sec CNT100;
   1:  PR[GP1:91,1] = PR[GP1:90,1] + 49.159;
   1:  PR[GP1:91,2] = PR[GP1:90,2] + 24.921;
   1:L PR[91] 10mm/sec CNT100;
   1:  PR[GP1:91,1] = PR[GP1:90,1] + 48.526;
   1:  PR[GP1:91,2] = PR[GP1:90,2] + 25.541;
   1:L PR[91] 10mm/sec CNT100;
   1:  PR[GP1:91,1] = PR[GP1:90,1] + 39.376;
   1:  PR[GP1:91,2] = PR[GP1:90,2] + 33.822;
   1:L PR[91] 10mm/sec CNT100;
   1:  PR[GP1:91,1] = PR[GP1:90,1] + 38.845;
   1:  PR[GP1:91,2] = PR[GP1:90,2] + 34.155;
   1:L PR[91] 10mm/sec CNT100;
   1:  PR[GP1:91,1] = PR[GP1:90,1] + 26.797;
   1:  PR[GP1:91,2] = PR[GP1:90,2] + 39.419;
   1:L PR[91] 10mm/sec CNT100;
   1:  PR[GP1:91,1] = PR[GP1:90,1] + 26.502;
   1:  PR[GP1:91,2] = PR[GP1:90,2] + 39.527;
   1:L PR[91] 10mm/sec CNT100;
   1:  PR[GP1:91,1] = PR[GP1:90,1] + 26.227;
   1:  PR[GP1:91,2] = PR[GP1:90,2] + 39.566;
   1:L PR[91] 10mm/sec CNT100;
   1:  PR[GP1:91,1] = PR[GP1:90,1] + 12.660;
   1:  PR[GP1:91,2] = PR[GP1:90,2] + 40.826;
   1:L PR[91] 10mm/sec CNT100;
   1:  PR[GP1:91,1] = PR[GP1:90,1] + -0.261;
   1:  PR[GP1:91,2] = PR[GP1:90,2] + 38.005;
   1:L PR[91] 10mm/sec CNT100;
   1:  PR[GP1:91,1] = PR[GP1:90,1] + -13.185;
   1:  PR[GP1:91,2] = PR[GP1:90,2] + 40.826;
   1:L PR[91] 10mm/sec CNT100;
   1:  PR[GP1:91,1] = PR[GP1:90,1] + -27.043;
   1:  PR[GP1:91,2] = PR[GP1:90,2] + 39.523;
   1:L PR[91] 10mm/sec CNT100;
   1:  PR[GP1:91,1] = PR[GP1:90,1] + -27.324;
   1:  PR[GP1:91,2] = PR[GP1:90,2] + 39.420;
   1:L PR[91] 10mm/sec CNT100;
   1:  PR[GP1:91,1] = PR[GP1:90,1] + -39.373;
   1:  PR[GP1:91,2] = PR[GP1:90,2] + 34.152;
   1:L PR[91] 10mm/sec CNT100;
   1:  PR[GP1:91,1] = PR[GP1:90,1] + -39.898;
   1:  PR[GP1:91,2] = PR[GP1:90,2] + 33.820;
   1:L PR[91] 10mm/sec CNT100;
   1:  PR[GP1:91,1] = PR[GP1:90,1] + -40.415;
   1:  PR[GP1:91,2] = PR[GP1:90,2] + 33.316;
   1:L PR[91] 10mm/sec CNT100;
   1:  PR[GP1:91,1] = PR[GP1:90,1] + -49.700;
   1:  PR[GP1:91,2] = PR[GP1:90,2] + 24.909;
   1:L PR[91] 10mm/sec CNT100;
   1:  PR[GP1:91,1] = PR[GP1:90,1] + -50.214;
   1:  PR[GP1:91,2] = PR[GP1:90,2] + 24.107;
   1:L PR[91] 10mm/sec CNT100;
   1:  PR[GP1:91,1] = PR[GP1:90,1] + -55.949;
   1:  PR[GP1:91,2] = PR[GP1:90,2] + 13.747;
   1:L PR[91] 10mm/sec CNT100;
   1:  PR[GP1:91,1] = PR[GP1:90,1] + -56.320;
   1:  PR[GP1:91,2] = PR[GP1:90,2] + 12.725;
   1:L PR[91] 10mm/sec CNT100;
   1:  PR[GP1:91,1] = PR[GP1:90,1] + -56.446;
   1:  PR[GP1:91,2] = PR[GP1:90,2] + 11.604;
   1:L PR[91] 10mm/sec CNT100;
   1:  PR[GP1:91,1] = PR[GP1:90,1] + -58.387;
   1:  PR[GP1:91,2] = PR[GP1:90,2] + 0.261;
   1:L PR[91] 10mm/sec CNT100;
   1:  PR[GP1:91,1] = PR[GP1:90,1] + -58.262;
   1:  PR[GP1:91,2] = PR[GP1:90,2] + -0.856;
   1:L PR[91] 10mm/sec CNT100;
   1:  PR[GP1:91,1] = PR[GP1:90,1] + -56.335;
   1:  PR[GP1:91,2] = PR[GP1:90,2] + -12.127;
   1:L PR[91] 10mm/sec CNT100;
   1:  PR[GP1:91,1] = PR[GP1:90,1] + -55.958;
   1:  PR[GP1:91,2] = PR[GP1:90,2] + -13.166;
   1:L PR[91] 10mm/sec CNT100;
   1:  PR[GP1:91,1] = PR[GP1:90,1] + -50.247;
   1:  PR[GP1:91,2] = PR[GP1:90,2] + -23.508;
   1:L PR[91] 10mm/sec CNT100;
   1:  PR[GP1:91,1] = PR[GP1:90,1] + -49.726;
   1:  PR[GP1:91,2] = PR[GP1:90,2] + -24.320;
   1:L PR[91] 10mm/sec CNT100;
   1:  PR[GP1:91,1] = PR[GP1:90,1] + -49.091;
   1:  PR[GP1:91,2] = PR[GP1:90,2] + -24.943;
   1:L PR[91] 10mm/sec CNT100;
   1:  PR[GP1:91,1] = PR[GP1:90,1] + -39.978;
   1:  PR[GP1:91,2] = PR[GP1:90,2] + -33.211;
   1:L PR[91] 10mm/sec CNT100;
   1:  PR[GP1:91,1] = PR[GP1:90,1] + -39.441;
   1:  PR[GP1:91,2] = PR[GP1:90,2] + -33.549;
   1:L PR[91] 10mm/sec CNT100;
   1:  PR[GP1:91,1] = PR[GP1:90,1] + -27.439;
   1:  PR[GP1:91,2] = PR[GP1:90,2] + -38.832;
   1:L PR[91] 10mm/sec CNT100;
   1:  PR[GP1:91,1] = PR[GP1:90,1] + -27.142;
   1:  PR[GP1:91,2] = PR[GP1:90,2] + -38.940;
   1:L PR[91] 10mm/sec CNT100;
   1:  PR[GP1:91,1] = PR[GP1:90,1] + -26.863;
   1:  PR[GP1:91,2] = PR[GP1:90,2] + -38.980;
   1:L PR[91] 10mm/sec CNT100;
   1:  PR[GP1:91,1] = PR[GP1:90,1] + -13.338;
   1:  PR[GP1:91,2] = PR[GP1:90,2] + -40.278;
   1:L PR[91] 10mm/sec CNT100;
   1:  PR[GP1:91,1] = PR[GP1:90,1] + -0.263;
   1:  PR[GP1:91,2] = PR[GP1:90,2] + -37.462;
   1:L PR[91] 10mm/sec CNT100;
   1:  PR[GP1:91,1] = PR[GP1:90,1] + 12.464;
   1:  PR[GP1:91,2] = PR[GP1:90,2] + -40.380;
   1:  PR[GP1:91,3] = PR[GP1:90,3] + 86.925;
   1:L PR[91] 10mm/sec CNT100;
   1:  PR[GP1:91,1] = PR[GP1:90,1] + 12.594;
   1:  PR[GP1:91,2] = PR[GP1:90,2] + -40.402;
   1:L PR[91] 10mm/sec CNT100;
   1:  PR[GP1:91,1] = PR[GP1:90,1] + 16.929;
   1:  PR[GP1:91,2] = PR[GP1:90,2] + -39.926;
   1:L PR[91] 10mm/sec CNT100;
   1:  PR[GP1:91,1] = PR[GP1:90,1] + 26.410;
   1:  PR[GP1:91,2] = PR[GP1:90,2] + -39.004;
   1:L PR[91] 10mm/sec CNT100;
   1:  PR[GP1:91,1] = PR[GP1:90,1] + 26.567;
   1:  PR[GP1:91,2] = PR[GP1:90,2] + -38.947;
   1:L PR[91] 10mm/sec CNT100;
   1:  PR[GP1:91,1] = PR[GP1:90,1] + 38.768;
   1:  PR[GP1:91,2] = PR[GP1:90,2] + -33.581;
   1:L PR[91] 10mm/sec CNT100;
   1:  PR[GP1:91,1] = PR[GP1:90,1] + 39.181;
   1:  PR[GP1:91,2] = PR[GP1:90,2] + -33.322;
   1:L PR[91] 10mm/sec CNT100;
   1:  PR[GP1:91,1] = PR[GP1:90,1] + 39.597;
   1:  PR[GP1:91,2] = PR[GP1:90,2] + -32.916;
   1:L PR[91] 10mm/sec CNT100;
   1:  PR[GP1:91,1] = PR[GP1:90,1] + 49.011;
   1:  PR[GP1:91,2] = PR[GP1:90,2] + -24.354;
   1:L PR[91] 10mm/sec CNT100;
   1:  PR[GP1:91,1] = PR[GP1:90,1] + 49.456;
   1:  PR[GP1:91,2] = PR[GP1:90,2] + -23.663;
   1:L PR[91] 10mm/sec CNT100;
   1:  PR[GP1:91,1] = PR[GP1:90,1] + 55.275;
   1:  PR[GP1:91,2] = PR[GP1:90,2] + -13.146;
   1:L PR[91] 10mm/sec CNT100;
   1:  PR[GP1:91,1] = PR[GP1:90,1] + 55.598;
   1:  PR[GP1:91,2] = PR[GP1:90,2] + -12.266;
   1:L PR[91] 10mm/sec CNT100;
   1:  PR[GP1:91,1] = PR[GP1:90,1] + 55.713;
   1:  PR[GP1:91,2] = PR[GP1:90,2] + -11.254;
   1:L PR[91] 10mm/sec CNT100;
   1:  PR[GP1:91,1] = PR[GP1:90,1] + 57.683;
   1:  PR[GP1:91,2] = PR[GP1:90,2] + 0.296;
   1:L PR[91] 10mm/sec CNT100;
   1:  PR[GP1:91,1] = PR[GP1:90,1] + 57.569;
   1:  PR[GP1:91,2] = PR[GP1:90,2] + 1.309;
   1:L PR[91] 10mm/sec CNT100;
   1:  PR[GP1:91,1] = PR[GP1:90,1] + 55.596;
   1:  PR[GP1:91,2] = PR[GP1:90,2] + 12.832;
   1:L PR[91] 10mm/sec CNT100;
   1:  PR[GP1:91,1] = PR[GP1:90,1] + 55.266;
   1:  PR[GP1:91,2] = PR[GP1:90,2] + 13.728;
   1:L PR[91] 10mm/sec CNT100;
   1:  PR[GP1:91,1] = PR[GP1:90,1] + 49.423;
   1:  PR[GP1:91,2] = PR[GP1:90,2] + 24.263;
   1:L PR[91] 10mm/sec CNT100;
   1:  PR[GP1:91,1] = PR[GP1:90,1] + 48.972;
   1:  PR[GP1:91,2] = PR[GP1:90,2] + 24.963;
   1:L PR[91] 10mm/sec CNT100;
   1:  PR[GP1:91,1] = PR[GP1:90,1] + 48.428;
   1:  PR[GP1:91,2] = PR[GP1:90,2] + 25.495;
   1:L PR[91] 10mm/sec CNT100;
   1:  PR[GP1:91,1] = PR[GP1:90,1] + 39.120;
   1:  PR[GP1:91,2] = PR[GP1:90,2] + 33.920;
   1:L PR[91] 10mm/sec CNT100;
   1:  PR[GP1:91,1] = PR[GP1:90,1] + 38.699;
   1:  PR[GP1:91,2] = PR[GP1:90,2] + 34.184;
   1:L PR[91] 10mm/sec CNT100;
   1:  PR[GP1:91,1] = PR[GP1:90,1] + 26.451;
   1:  PR[GP1:91,2] = PR[GP1:90,2] + 39.535;
   1:L PR[91] 10mm/sec CNT100;
   1:  PR[GP1:91,1] = PR[GP1:90,1] + 26.283;
   1:  PR[GP1:91,2] = PR[GP1:90,2] + 39.597;
   1:L PR[91] 10mm/sec CNT100;
   1:  PR[GP1:91,1] = PR[GP1:90,1] + 26.128;
   1:  PR[GP1:91,2] = PR[GP1:90,2] + 39.619;
   1:L PR[91] 10mm/sec CNT100;
   1:  PR[GP1:91,1] = PR[GP1:90,1] + 16.931;
   1:  PR[GP1:91,2] = PR[GP1:90,2] + 40.473;
   1:L PR[91] 10mm/sec CNT100;
   1:  PR[GP1:91,1] = PR[GP1:90,1] + 12.449;
   1:  PR[GP1:91,2] = PR[GP1:90,2] + 40.952;
   1:L PR[91] 10mm/sec CNT100;
   1:  PR[GP1:91,1] = PR[GP1:90,1] + 12.219;
   1:  PR[GP1:91,2] = PR[GP1:90,2] + 40.912;
   1:L PR[91] 10mm/sec CNT100;
   1:  PR[GP1:91,1] = PR[GP1:90,1] + -0.261;
   1:  PR[GP1:91,2] = PR[GP1:90,2] + 38.189;
   1:L PR[91] 10mm/sec CNT100;
   1:  PR[GP1:91,1] = PR[GP1:90,1] + -12.744;
   1:  PR[GP1:91,2] = PR[GP1:90,2] + 40.911;
   1:L PR[91] 10mm/sec CNT100;
   1:  PR[GP1:91,1] = PR[GP1:90,1] + -12.975;
   1:  PR[GP1:91,2] = PR[GP1:90,2] + 40.952;
   1:L PR[91] 10mm/sec CNT100;
   1:  PR[GP1:91,1] = PR[GP1:90,1] + -17.456;
   1:  PR[GP1:91,2] = PR[GP1:90,2] + 40.474;
   1:L PR[91] 10mm/sec CNT100;
   1:  PR[GP1:91,1] = PR[GP1:90,1] + -26.823;
   1:  PR[GP1:91,2] = PR[GP1:90,2] + 39.593;
   1:L PR[91] 10mm/sec CNT100;
   1:  PR[GP1:91,1] = PR[GP1:90,1] + -26.978;
   1:  PR[GP1:91,2] = PR[GP1:90,2] + 39.536;
   1:L PR[91] 10mm/sec CNT100;
   1:  PR[GP1:91,1] = PR[GP1:90,1] + -39.226;
   1:  PR[GP1:91,2] = PR[GP1:90,2] + 34.181;
   1:L PR[91] 10mm/sec CNT100;
   1:  PR[GP1:91,1] = PR[GP1:90,1] + -39.641;
   1:  PR[GP1:91,2] = PR[GP1:90,2] + 33.920;
   1:L PR[91] 10mm/sec CNT100;
   1:  PR[GP1:91,1] = PR[GP1:90,1] + -40.057;
   1:  PR[GP1:91,2] = PR[GP1:90,2] + 33.513;
   1:L PR[91] 10mm/sec CNT100;
   1:  PR[GP1:91,1] = PR[GP1:90,1] + -49.511;
   1:  PR[GP1:91,2] = PR[GP1:90,2] + 24.953;
   1:L PR[91] 10mm/sec CNT100;
   1:  PR[GP1:91,1] = PR[GP1:90,1] + -49.951;
   1:  PR[GP1:91,2] = PR[GP1:90,2] + 24.267;
   1:L PR[91] 10mm/sec CNT100;
   1:  PR[GP1:91,1] = PR[GP1:90,1] + -55.795;
   1:  PR[GP1:91,2] = PR[GP1:90,2] + 13.711;
   1:L PR[91] 10mm/sec CNT100;
   1:  PR[GP1:91,1] = PR[GP1:90,1] + -56.120;
   1:  PR[GP1:91,2] = PR[GP1:90,2] + 12.815;
   1:L PR[91] 10mm/sec CNT100;
   1:  PR[GP1:91,1] = PR[GP1:90,1] + -56.231;
   1:  PR[GP1:91,2] = PR[GP1:90,2] + 11.824;
   1:L PR[91] 10mm/sec CNT100;
   1:  PR[GP1:91,1] = PR[GP1:90,1] + -58.210;
   1:  PR[GP1:91,2] = PR[GP1:90,2] + 0.261;
   1:L PR[91] 10mm/sec CNT100;
   1:  PR[GP1:91,1] = PR[GP1:90,1] + -58.099;
   1:  PR[GP1:91,2] = PR[GP1:90,2] + -0.728;
   1:L PR[91] 10mm/sec CNT100;
   1:  PR[GP1:91,1] = PR[GP1:90,1] + -56.135;
   1:  PR[GP1:91,2] = PR[GP1:90,2] + -12.216;
   1:L PR[91] 10mm/sec CNT100;
   1:  PR[GP1:91,1] = PR[GP1:90,1] + -55.803;
   1:  PR[GP1:91,2] = PR[GP1:90,2] + -13.130;
   1:L PR[91] 10mm/sec CNT100;
   1:  PR[GP1:91,1] = PR[GP1:90,1] + -49.985;
   1:  PR[GP1:91,2] = PR[GP1:90,2] + -23.666;
   1:L PR[91] 10mm/sec CNT100;
   1:  PR[GP1:91,1] = PR[GP1:90,1] + -49.538;
   1:  PR[GP1:91,2] = PR[GP1:90,2] + -24.363;
   1:L PR[91] 10mm/sec CNT100;
   1:  PR[GP1:91,1] = PR[GP1:90,1] + -48.994;
   1:  PR[GP1:91,2] = PR[GP1:90,2] + -24.897;
   1:L PR[91] 10mm/sec CNT100;
   1:  PR[GP1:91,1] = PR[GP1:90,1] + -39.721;
   1:  PR[GP1:91,2] = PR[GP1:90,2] + -33.309;
   1:L PR[91] 10mm/sec CNT100;
   1:  PR[GP1:91,1] = PR[GP1:90,1] + -39.295;
   1:  PR[GP1:91,2] = PR[GP1:90,2] + -33.578;
   1:L PR[91] 10mm/sec CNT100;
   1:  PR[GP1:91,1] = PR[GP1:90,1] + -27.094;
   1:  PR[GP1:91,2] = PR[GP1:90,2] + -38.948;
   1:L PR[91] 10mm/sec CNT100;
   1:  PR[GP1:91,1] = PR[GP1:90,1] + -26.924;
   1:  PR[GP1:91,2] = PR[GP1:90,2] + -39.010;
   1:L PR[91] 10mm/sec CNT100;
   1:  PR[GP1:91,1] = PR[GP1:90,1] + -26.765;
   1:  PR[GP1:91,2] = PR[GP1:90,2] + -39.033;
   1:L PR[91] 10mm/sec CNT100;
   1:  PR[GP1:91,1] = PR[GP1:90,1] + -17.458;
   1:  PR[GP1:91,2] = PR[GP1:90,2] + -39.926;
   1:L PR[91] 10mm/sec CNT100;
   1:  PR[GP1:91,1] = PR[GP1:90,1] + -13.120;
   1:  PR[GP1:91,2] = PR[GP1:90,2] + -40.402;
   1:L PR[91] 10mm/sec CNT100;
   1:  PR[GP1:91,1] = PR[GP1:90,1] + -12.990;
   1:  PR[GP1:91,2] = PR[GP1:90,2] + -40.380;
   1:L PR[91] 10mm/sec CNT100;
   1:  PR[GP1:91,1] = PR[GP1:90,1] + -0.263;
   1:  PR[GP1:91,2] = PR[GP1:90,2] + -37.643;
   1:L PR[91] 10mm/sec CNT100;
   1:  PR[GP1:91,1] = PR[GP1:90,1] + 12.026;
   1:  PR[GP1:91,2] = PR[GP1:90,2] + -40.467;
   1:  PR[GP1:91,3] = PR[GP1:90,3] + 87.535;
   1:L PR[91] 10mm/sec CNT100;
   1:  PR[GP1:91,1] = PR[GP1:90,1] + 12.404;
   1:  PR[GP1:91,2] = PR[GP1:90,2] + -40.530;
   1:L PR[91] 10mm/sec CNT100;
   1:  PR[GP1:91,1] = PR[GP1:90,1] + 21.601;
   1:  PR[GP1:91,2] = PR[GP1:90,2] + -39.520;
   1:L PR[91] 10mm/sec CNT100;
   1:  PR[GP1:91,1] = PR[GP1:90,1] + 26.173;
   1:  PR[GP1:91,2] = PR[GP1:90,2] + -39.076;
   1:L PR[91] 10mm/sec CNT100;
   1:  PR[GP1:91,1] = PR[GP1:90,1] + 38.623;
   1:  PR[GP1:91,2] = PR[GP1:90,2] + -33.610;
   1:L PR[91] 10mm/sec CNT100;
   1:  PR[GP1:91,1] = PR[GP1:90,1] + 38.925;
   1:  PR[GP1:91,2] = PR[GP1:90,2] + -33.420;
   1:L PR[91] 10mm/sec CNT100;
   1:  PR[GP1:91,1] = PR[GP1:90,1] + 39.242;
   1:  PR[GP1:91,2] = PR[GP1:90,2] + -33.111;
   1:L PR[91] 10mm/sec CNT100;
   1:  PR[GP1:91,1] = PR[GP1:90,1] + 48.824;
   1:  PR[GP1:91,2] = PR[GP1:90,2] + -24.396;
   1:L PR[91] 10mm/sec CNT100;
   1:  PR[GP1:91,1] = PR[GP1:90,1] + 49.194;
   1:  PR[GP1:91,2] = PR[GP1:90,2] + -23.821;
   1:L PR[91] 10mm/sec CNT100;
   1:  PR[GP1:91,1] = PR[GP1:90,1] + 55.120;
   1:  PR[GP1:91,2] = PR[GP1:90,2] + -13.109;
   1:L PR[91] 10mm/sec CNT100;
   1:  PR[GP1:91,1] = PR[GP1:90,1] + 55.399;
   1:  PR[GP1:91,2] = PR[GP1:90,2] + -12.353;
   1:L PR[91] 10mm/sec CNT100;
   1:  PR[GP1:91,1] = PR[GP1:90,1] + 55.499;
   1:  PR[GP1:91,2] = PR[GP1:90,2] + -11.474;
   1:L PR[91] 10mm/sec CNT100;
   1:  PR[GP1:91,1] = PR[GP1:90,1] + 57.506;
   1:  PR[GP1:91,2] = PR[GP1:90,2] + 0.296;
   1:L PR[91] 10mm/sec CNT100;
   1:  PR[GP1:91,1] = PR[GP1:90,1] + 57.406;
   1:  PR[GP1:91,2] = PR[GP1:90,2] + 1.179;
   1:L PR[91] 10mm/sec CNT100;
   1:  PR[GP1:91,1] = PR[GP1:90,1] + 55.396;
   1:  PR[GP1:91,2] = PR[GP1:90,2] + 12.919;
   1:L PR[91] 10mm/sec CNT100;
   1:  PR[GP1:91,1] = PR[GP1:90,1] + 55.112;
   1:  PR[GP1:91,2] = PR[GP1:90,2] + 13.691;
   1:L PR[91] 10mm/sec CNT100;
   1:  PR[GP1:91,1] = PR[GP1:90,1] + 49.161;
   1:  PR[GP1:91,2] = PR[GP1:90,2] + 24.422;
   1:L PR[91] 10mm/sec CNT100;
   1:  PR[GP1:91,1] = PR[GP1:90,1] + 48.784;
   1:  PR[GP1:91,2] = PR[GP1:90,2] + 25.006;
   1:L PR[91] 10mm/sec CNT100;
   1:  PR[GP1:91,1] = PR[GP1:90,1] + 48.331;
   1:  PR[GP1:91,2] = PR[GP1:90,2] + 25.449;
   1:L PR[91] 10mm/sec CNT100;
   1:  PR[GP1:91,1] = PR[GP1:90,1] + 38.863;
   1:  PR[GP1:91,2] = PR[GP1:90,2] + 34.019;
   1:L PR[91] 10mm/sec CNT100;
   1:  PR[GP1:91,1] = PR[GP1:90,1] + 38.552;
   1:  PR[GP1:91,2] = PR[GP1:90,2] + 34.213;
   1:L PR[91] 10mm/sec CNT100;
   1:  PR[GP1:91,1] = PR[GP1:90,1] + 26.105;
   1:  PR[GP1:91,2] = PR[GP1:90,2] + 39.652;
   1:L PR[91] 10mm/sec CNT100;
   1:  PR[GP1:91,1] = PR[GP1:90,1] + 26.064;
   1:  PR[GP1:91,2] = PR[GP1:90,2] + 39.667;
   1:L PR[91] 10mm/sec CNT100;
   1:  PR[GP1:91,1] = PR[GP1:90,1] + 26.029;
   1:  PR[GP1:91,2] = PR[GP1:90,2] + 39.672;
   1:L PR[91] 10mm/sec CNT100;
   1:  PR[GP1:91,1] = PR[GP1:90,1] + 21.603;
   1:  PR[GP1:91,2] = PR[GP1:90,2] + 40.083;
   1:L PR[91] 10mm/sec CNT100;
   1:  PR[GP1:91,1] = PR[GP1:90,1] + 12.262;
   1:  PR[GP1:91,2] = PR[GP1:90,2] + 41.081;
   1:L PR[91] 10mm/sec CNT100;
   1:  PR[GP1:91,1] = PR[GP1:90,1] + 11.686;
   1:  PR[GP1:91,2] = PR[GP1:90,2] + 40.979;
   1:L PR[91] 10mm/sec CNT100;
   1:  PR[GP1:91,1] = PR[GP1:90,1] + -0.261;
   1:  PR[GP1:91,2] = PR[GP1:90,2] + 38.373;
   1:L PR[91] 10mm/sec CNT100;
   1:  PR[GP1:91,1] = PR[GP1:90,1] + -12.211;
   1:  PR[GP1:91,2] = PR[GP1:90,2] + 40.979;
   1:L PR[91] 10mm/sec CNT100;
   1:  PR[GP1:91,1] = PR[GP1:90,1] + -12.788;
   1:  PR[GP1:91,2] = PR[GP1:90,2] + 41.080;
   1:L PR[91] 10mm/sec CNT100;
   1:  PR[GP1:91,1] = PR[GP1:90,1] + -22.128;
   1:  PR[GP1:91,2] = PR[GP1:90,2] + 40.084;
   1:L PR[91] 10mm/sec CNT100;
   1:  PR[GP1:91,1] = PR[GP1:90,1] + -26.585;
   1:  PR[GP1:91,2] = PR[GP1:90,2] + 39.665;
   1:L PR[91] 10mm/sec CNT100;
   1:  PR[GP1:91,1] = PR[GP1:90,1] + -39.079;
   1:  PR[GP1:91,2] = PR[GP1:90,2] + 34.210;
   1:L PR[91] 10mm/sec CNT100;
   1:  PR[GP1:91,1] = PR[GP1:90,1] + -39.383;
   1:  PR[GP1:91,2] = PR[GP1:90,2] + 34.019;
   1:L PR[91] 10mm/sec CNT100;
   1:  PR[GP1:91,1] = PR[GP1:90,1] + -39.700;
   1:  PR[GP1:91,2] = PR[GP1:90,2] + 33.709;
   1:L PR[91] 10mm/sec CNT100;
   1:  PR[GP1:91,1] = PR[GP1:90,1] + -49.323;
   1:  PR[GP1:91,2] = PR[GP1:90,2] + 24.997;
   1:L PR[91] 10mm/sec CNT100;
   1:  PR[GP1:91,1] = PR[GP1:90,1] + -49.688;
   1:  PR[GP1:91,2] = PR[GP1:90,2] + 24.426;
   1:L PR[91] 10mm/sec CNT100;
   1:  PR[GP1:91,1] = PR[GP1:90,1] + -55.640;
   1:  PR[GP1:91,2] = PR[GP1:90,2] + 13.675;
   1:L PR[91] 10mm/sec CNT100;
   1:  PR[GP1:91,1] = PR[GP1:90,1] + -55.920;
   1:  PR[GP1:91,2] = PR[GP1:90,2] + 12.905;
   1:L PR[91] 10mm/sec CNT100;
   1:  PR[GP1:91,1] = PR[GP1:90,1] + -56.016;
   1:  PR[GP1:91,2] = PR[GP1:90,2] + 12.044;
   1:L PR[91] 10mm/sec CNT100;
   1:  PR[GP1:91,1] = PR[GP1:90,1] + -58.032;
   1:  PR[GP1:91,2] = PR[GP1:90,2] + 0.261;
   1:L PR[91] 10mm/sec CNT100;
   1:  PR[GP1:91,1] = PR[GP1:90,1] + -57.936;
   1:  PR[GP1:91,2] = PR[GP1:90,2] + -0.600;
   1:L PR[91] 10mm/sec CNT100;
   1:  PR[GP1:91,1] = PR[GP1:90,1] + -55.934;
   1:  PR[GP1:91,2] = PR[GP1:90,2] + -12.306;
   1:L PR[91] 10mm/sec CNT100;
   1:  PR[GP1:91,1] = PR[GP1:90,1] + -55.649;
   1:  PR[GP1:91,2] = PR[GP1:90,2] + -13.093;
   1:L PR[91] 10mm/sec CNT100;
   1:  PR[GP1:91,1] = PR[GP1:90,1] + -49.722;
   1:  PR[GP1:91,2] = PR[GP1:90,2] + -23.825;
   1:L PR[91] 10mm/sec CNT100;
   1:  PR[GP1:91,1] = PR[GP1:90,1] + -49.350;
   1:  PR[GP1:91,2] = PR[GP1:90,2] + -24.406;
   1:L PR[91] 10mm/sec CNT100;
   1:  PR[GP1:91,1] = PR[GP1:90,1] + -48.896;
   1:  PR[GP1:91,2] = PR[GP1:90,2] + -24.852;
   1:L PR[91] 10mm/sec CNT100;
   1:  PR[GP1:91,1] = PR[GP1:90,1] + -39.464;
   1:  PR[GP1:91,2] = PR[GP1:90,2] + -33.408;
   1:L PR[91] 10mm/sec CNT100;
   1:  PR[GP1:91,1] = PR[GP1:90,1] + -39.150;
   1:  PR[GP1:91,2] = PR[GP1:90,2] + -33.606;
   1:L PR[91] 10mm/sec CNT100;
   1:  PR[GP1:91,1] = PR[GP1:90,1] + -26.700;
   1:  PR[GP1:91,2] = PR[GP1:90,2] + -39.077;
   1:L PR[91] 10mm/sec CNT100;
   1:  PR[GP1:91,1] = PR[GP1:90,1] + -22.129;
   1:  PR[GP1:91,2] = PR[GP1:90,2] + -39.521;
   1:L PR[91] 10mm/sec CNT100;
   1:  PR[GP1:91,1] = PR[GP1:90,1] + -12.931;
   1:  PR[GP1:91,2] = PR[GP1:90,2] + -40.530;
   1:L PR[91] 10mm/sec CNT100;
   1:  PR[GP1:91,1] = PR[GP1:90,1] + -12.552;
   1:  PR[GP1:91,2] = PR[GP1:90,2] + -40.466;
   1:L PR[91] 10mm/sec CNT100;
   1:  PR[GP1:91,1] = PR[GP1:90,1] + -0.263;
   1:  PR[GP1:91,2] = PR[GP1:90,2] + -37.824;
   1:L PR[91] 10mm/sec CNT100;
   1:  PR[GP1:91,1] = PR[GP1:90,1] + 11.588;
   1:  PR[GP1:91,2] = PR[GP1:90,2] + -40.554;
   1:  PR[GP1:91,3] = PR[GP1:90,3] + 88.145;
   1:L PR[91] 10mm/sec CNT100;
   1:  PR[GP1:91,1] = PR[GP1:90,1] + 12.215;
   1:  PR[GP1:91,2] = PR[GP1:90,2] + -40.659;
   1:L PR[91] 10mm/sec CNT100;
   1:  PR[GP1:91,1] = PR[GP1:90,1] + 25.956;
   1:  PR[GP1:91,2] = PR[GP1:90,2] + -39.148;
   1:L PR[91] 10mm/sec CNT100;
   1:  PR[GP1:91,1] = PR[GP1:90,1] + 38.477;
   1:  PR[GP1:91,2] = PR[GP1:90,2] + -33.638;
   1:L PR[91] 10mm/sec CNT100;
   1:  PR[GP1:91,1] = PR[GP1:90,1] + 38.670;
   1:  PR[GP1:91,2] = PR[GP1:90,2] + -33.517;
   1:L PR[91] 10mm/sec CNT100;
   1:  PR[GP1:91,1] = PR[GP1:90,1] + 38.887;
   1:  PR[GP1:91,2] = PR[GP1:90,2] + -33.305;
   1:L PR[91] 10mm/sec CNT100;
   1:  PR[GP1:91,1] = PR[GP1:90,1] + 48.637;
   1:  PR[GP1:91,2] = PR[GP1:90,2] + -24.437;
   1:L PR[91] 10mm/sec CNT100;
   1:  PR[GP1:91,1] = PR[GP1:90,1] + 48.933;
   1:  PR[GP1:91,2] = PR[GP1:90,2] + -23.978;
   1:L PR[91] 10mm/sec CNT100;
   1:  PR[GP1:91,1] = PR[GP1:90,1] + 54.966;
   1:  PR[GP1:91,2] = PR[GP1:90,2] + -13.072;
   1:L PR[91] 10mm/sec CNT100;
   1:  PR[GP1:91,1] = PR[GP1:90,1] + 55.199;
   1:  PR[GP1:91,2] = PR[GP1:90,2] + -12.440;
   1:L PR[91] 10mm/sec CNT100;
   1:  PR[GP1:91,1] = PR[GP1:90,1] + 55.284;
   1:  PR[GP1:91,2] = PR[GP1:90,2] + -11.693;
   1:L PR[91] 10mm/sec CNT100;
   1:  PR[GP1:91,1] = PR[GP1:90,1] + 57.329;
   1:  PR[GP1:91,2] = PR[GP1:90,2] + 0.296;
   1:L PR[91] 10mm/sec CNT100;
   1:  PR[GP1:91,1] = PR[GP1:90,1] + 57.244;
   1:  PR[GP1:91,2] = PR[GP1:90,2] + 1.048;
   1:L PR[91] 10mm/sec CNT100;
   1:  PR[GP1:91,1] = PR[GP1:90,1] + 55.196;
   1:  PR[GP1:91,2] = PR[GP1:90,2] + 13.006;
   1:L PR[91] 10mm/sec CNT100;
   1:  PR[GP1:91,1] = PR[GP1:90,1] + 54.958;
   1:  PR[GP1:91,2] = PR[GP1:90,2] + 13.655;
   1:L PR[91] 10mm/sec CNT100;
   1:  PR[GP1:91,1] = PR[GP1:90,1] + 48.898;
   1:  PR[GP1:91,2] = PR[GP1:90,2] + 24.580;
   1:L PR[91] 10mm/sec CNT100;
   1:  PR[GP1:91,1] = PR[GP1:90,1] + 48.597;
   1:  PR[GP1:91,2] = PR[GP1:90,2] + 25.048;
   1:L PR[91] 10mm/sec CNT100;
   1:  PR[GP1:91,1] = PR[GP1:90,1] + 48.234;
   1:  PR[GP1:91,2] = PR[GP1:90,2] + 25.403;
   1:L PR[91] 10mm/sec CNT100;
   1:  PR[GP1:91,1] = PR[GP1:90,1] + 38.606;
   1:  PR[GP1:91,2] = PR[GP1:90,2] + 34.117;
   1:L PR[91] 10mm/sec CNT100;
   1:  PR[GP1:91,1] = PR[GP1:90,1] + 38.406;
   1:  PR[GP1:91,2] = PR[GP1:90,2] + 34.242;
   1:L PR[91] 10mm/sec CNT100;
   1:  PR[GP1:91,1] = PR[GP1:90,1] + 25.823;
   1:  PR[GP1:91,2] = PR[GP1:90,2] + 39.741;
   1:L PR[91] 10mm/sec CNT100;
   1:  PR[GP1:91,1] = PR[GP1:90,1] + 12.075;
   1:  PR[GP1:91,2] = PR[GP1:90,2] + 41.209;
   1:L PR[91] 10mm/sec CNT100;
   1:  PR[GP1:91,1] = PR[GP1:90,1] + 11.152;
   1:  PR[GP1:91,2] = PR[GP1:90,2] + 41.047;
   1:L PR[91] 10mm/sec CNT100;
   1:  PR[GP1:91,1] = PR[GP1:90,1] + -0.260;
   1:  PR[GP1:91,2] = PR[GP1:90,2] + 38.557;
   1:L PR[91] 10mm/sec CNT100;
   1:  PR[GP1:91,1] = PR[GP1:90,1] + -11.677;
   1:  PR[GP1:91,2] = PR[GP1:90,2] + 41.046;
   1:L PR[91] 10mm/sec CNT100;
   1:  PR[GP1:91,1] = PR[GP1:90,1] + -12.600;
   1:  PR[GP1:91,2] = PR[GP1:90,2] + 41.209;
   1:L PR[91] 10mm/sec CNT100;
   1:  PR[GP1:91,1] = PR[GP1:90,1] + -26.368;
   1:  PR[GP1:91,2] = PR[GP1:90,2] + 39.739;
   1:L PR[91] 10mm/sec CNT100;
   1:  PR[GP1:91,1] = PR[GP1:90,1] + -38.932;
   1:  PR[GP1:91,2] = PR[GP1:90,2] + 34.240;
   1:L PR[91] 10mm/sec CNT100;
   1:  PR[GP1:91,1] = PR[GP1:90,1] + -39.125;
   1:  PR[GP1:91,2] = PR[GP1:90,2] + 34.118;
   1:L PR[91] 10mm/sec CNT100;
   1:  PR[GP1:91,1] = PR[GP1:90,1] + -39.342;
   1:  PR[GP1:91,2] = PR[GP1:90,2] + 33.906;
   1:L PR[91] 10mm/sec CNT100;
   1:  PR[GP1:91,1] = PR[GP1:90,1] + -49.134;
   1:  PR[GP1:91,2] = PR[GP1:90,2] + 25.040;
   1:L PR[91] 10mm/sec CNT100;
   1:  PR[GP1:91,1] = PR[GP1:90,1] + -49.426;
   1:  PR[GP1:91,2] = PR[GP1:90,2] + 24.585;
   1:L PR[91] 10mm/sec CNT100;
   1:  PR[GP1:91,1] = PR[GP1:90,1] + -55.485;
   1:  PR[GP1:91,2] = PR[GP1:90,2] + 13.639;
   1:L PR[91] 10mm/sec CNT100;
   1:  PR[GP1:91,1] = PR[GP1:90,1] + -55.719;
   1:  PR[GP1:91,2] = PR[GP1:90,2] + 12.995;
   1:L PR[91] 10mm/sec CNT100;
   1:  PR[GP1:91,1] = PR[GP1:90,1] + -55.801;
   1:  PR[GP1:91,2] = PR[GP1:90,2] + 12.264;
   1:L PR[91] 10mm/sec CNT100;
   1:  PR[GP1:91,1] = PR[GP1:90,1] + -57.855;
   1:  PR[GP1:91,2] = PR[GP1:90,2] + 0.261;
   1:L PR[91] 10mm/sec CNT100;
   1:  PR[GP1:91,1] = PR[GP1:90,1] + -57.773;
   1:  PR[GP1:91,2] = PR[GP1:90,2] + -0.472;
   1:L PR[91] 10mm/sec CNT100;
   1:  PR[GP1:91,1] = PR[GP1:90,1] + -55.734;
   1:  PR[GP1:91,2] = PR[GP1:90,2] + -12.395;
   1:L PR[91] 10mm/sec CNT100;
   1:  PR[GP1:91,1] = PR[GP1:90,1] + -55.494;
   1:  PR[GP1:91,2] = PR[GP1:90,2] + -13.057;
   1:L PR[91] 10mm/sec CNT100;
   1:  PR[GP1:91,1] = PR[GP1:90,1] + -49.460;
   1:  PR[GP1:91,2] = PR[GP1:90,2] + -23.983;
   1:L PR[91] 10mm/sec CNT100;
   1:  PR[GP1:91,1] = PR[GP1:90,1] + -49.162;
   1:  PR[GP1:91,2] = PR[GP1:90,2] + -24.449;
   1:L PR[91] 10mm/sec CNT100;
   1:  PR[GP1:91,1] = PR[GP1:90,1] + -48.798;
   1:  PR[GP1:91,2] = PR[GP1:90,2] + -24.806;
   1:L PR[91] 10mm/sec CNT100;
   1:  PR[GP1:91,1] = PR[GP1:90,1] + -39.208;
   1:  PR[GP1:91,2] = PR[GP1:90,2] + -33.506;
   1:L PR[91] 10mm/sec CNT100;
   1:  PR[GP1:91,1] = PR[GP1:90,1] + -39.004;
   1:  PR[GP1:91,2] = PR[GP1:90,2] + -33.635;
   1:L PR[91] 10mm/sec CNT100;
   1:  PR[GP1:91,1] = PR[GP1:90,1] + -26.482;
   1:  PR[GP1:91,2] = PR[GP1:90,2] + -39.150;
   1:L PR[91] 10mm/sec CNT100;
   1:  PR[GP1:91,1] = PR[GP1:90,1] + -12.742;
   1:  PR[GP1:91,2] = PR[GP1:90,2] + -40.658;
   1:L PR[91] 10mm/sec CNT100;
   1:  PR[GP1:91,1] = PR[GP1:90,1] + -12.113;
   1:  PR[GP1:91,2] = PR[GP1:90,2] + -40.553;
   1:L PR[91] 10mm/sec CNT100;
   1:  PR[GP1:91,1] = PR[GP1:90,1] + -0.263;
   1:  PR[GP1:91,2] = PR[GP1:90,2] + -38.005;
   1:L PR[91] 10mm/sec CNT100;
   1:  PR[GP1:91,1] = PR[GP1:90,1] + 11.150;
   1:  PR[GP1:91,2] = PR[GP1:90,2] + -40.640;
   1:  PR[GP1:91,3] = PR[GP1:90,3] + 88.755;
   1:L PR[91] 10mm/sec CNT100;
   1:  PR[GP1:91,1] = PR[GP1:90,1] + 12.026;
   1:  PR[GP1:91,2] = PR[GP1:90,2] + -40.787;
   1:L PR[91] 10mm/sec CNT100;
   1:  PR[GP1:91,1] = PR[GP1:90,1] + 25.612;
   1:  PR[GP1:91,2] = PR[GP1:90,2] + -39.295;
   1:L PR[91] 10mm/sec CNT100;
   1:  PR[GP1:91,1] = PR[GP1:90,1] + 25.804;
   1:  PR[GP1:91,2] = PR[GP1:90,2] + -39.259;
   1:L PR[91] 10mm/sec CNT100;
   1:  PR[GP1:91,1] = PR[GP1:90,1] + 30.774;
   1:  PR[GP1:91,2] = PR[GP1:90,2] + -36.990;
   1:L PR[91] 10mm/sec CNT100;
   1:  PR[GP1:91,1] = PR[GP1:90,1] + 38.332;
   1:  PR[GP1:91,2] = PR[GP1:90,2] + -33.666;
   1:L PR[91] 10mm/sec CNT100;
   1:  PR[GP1:91,1] = PR[GP1:90,1] + 38.423;
   1:  PR[GP1:91,2] = PR[GP1:90,2] + -33.609;
   1:L PR[91] 10mm/sec CNT100;
   1:  PR[GP1:91,1] = PR[GP1:90,1] + 48.450;
   1:  PR[GP1:91,2] = PR[GP1:90,2] + -24.479;
   1:L PR[91] 10mm/sec CNT100;
   1:  PR[GP1:91,1] = PR[GP1:90,1] + 48.671;
   1:  PR[GP1:91,2] = PR[GP1:90,2] + -24.136;
   1:L PR[91] 10mm/sec CNT100;
   1:  PR[GP1:91,1] = PR[GP1:90,1] + 54.812;
   1:  PR[GP1:91,2] = PR[GP1:90,2] + -13.036;
   1:L PR[91] 10mm/sec CNT100;
   1:  PR[GP1:91,1] = PR[GP1:90,1] + 54.999;
   1:  PR[GP1:91,2] = PR[GP1:90,2] + -12.526;
   1:L PR[91] 10mm/sec CNT100;
   1:  PR[GP1:91,1] = PR[GP1:90,1] + 55.069;
   1:  PR[GP1:91,2] = PR[GP1:90,2] + -11.913;
   1:L PR[91] 10mm/sec CNT100;
   1:  PR[GP1:91,1] = PR[GP1:90,1] + 57.152;
   1:  PR[GP1:91,2] = PR[GP1:90,2] + 0.296;
   1:L PR[91] 10mm/sec CNT100;
   1:  PR[GP1:91,1] = PR[GP1:90,1] + 57.081;
   1:  PR[GP1:91,2] = PR[GP1:90,2] + 0.917;
   1:L PR[91] 10mm/sec CNT100;
   1:  PR[GP1:91,1] = PR[GP1:90,1] + 54.996;
   1:  PR[GP1:91,2] = PR[GP1:90,2] + 13.094;
   1:L PR[91] 10mm/sec CNT100;
   1:  PR[GP1:91,1] = PR[GP1:90,1] + 54.803;
   1:  PR[GP1:91,2] = PR[GP1:90,2] + 13.618;
   1:L PR[91] 10mm/sec CNT100;
   1:  PR[GP1:91,1] = PR[GP1:90,1] + 48.636;
   1:  PR[GP1:91,2] = PR[GP1:90,2] + 24.738;
   1:L PR[91] 10mm/sec CNT100;
   1:  PR[GP1:91,1] = PR[GP1:90,1] + 48.409;
   1:  PR[GP1:91,2] = PR[GP1:90,2] + 25.090;
   1:L PR[91] 10mm/sec CNT100;
   1:  PR[GP1:91,1] = PR[GP1:90,1] + 48.136;
   1:  PR[GP1:91,2] = PR[GP1:90,2] + 25.358;
   1:L PR[91] 10mm/sec CNT100;
   1:  PR[GP1:91,1] = PR[GP1:90,1] + 38.349;
   1:  PR[GP1:91,2] = PR[GP1:90,2] + 34.215;
   1:L PR[91] 10mm/sec CNT100;
   1:  PR[GP1:91,1] = PR[GP1:90,1] + 38.260;
   1:  PR[GP1:91,2] = PR[GP1:90,2] + 34.271;
   1:L PR[91] 10mm/sec CNT100;
   1:  PR[GP1:91,1] = PR[GP1:90,1] + 30.775;
   1:  PR[GP1:91,2] = PR[GP1:90,2] + 37.541;
   1:L PR[91] 10mm/sec CNT100;
   1:  PR[GP1:91,1] = PR[GP1:90,1] + 25.692;
   1:  PR[GP1:91,2] = PR[GP1:90,2] + 39.848;
   1:L PR[91] 10mm/sec CNT100;
   1:  PR[GP1:91,1] = PR[GP1:90,1] + 25.493;
   1:  PR[GP1:91,2] = PR[GP1:90,2] + 39.885;
   1:L PR[91] 10mm/sec CNT100;
   1:  PR[GP1:91,1] = PR[GP1:90,1] + 11.887;
   1:  PR[GP1:91,2] = PR[GP1:90,2] + 41.338;
   1:L PR[91] 10mm/sec CNT100;
   1:  PR[GP1:91,1] = PR[GP1:90,1] + 10.619;
   1:  PR[GP1:91,2] = PR[GP1:90,2] + 41.115;
   1:L PR[91] 10mm/sec CNT100;
   1:  PR[GP1:91,1] = PR[GP1:90,1] + -0.260;
   1:  PR[GP1:91,2] = PR[GP1:90,2] + 38.742;
   1:L PR[91] 10mm/sec CNT100;
   1:  PR[GP1:91,1] = PR[GP1:90,1] + -11.143;
   1:  PR[GP1:91,2] = PR[GP1:90,2] + 41.114;
   1:L PR[91] 10mm/sec CNT100;
   1:  PR[GP1:91,1] = PR[GP1:90,1] + -12.413;
   1:  PR[GP1:91,2] = PR[GP1:90,2] + 41.337;
   1:L PR[91] 10mm/sec CNT100;
   1:  PR[GP1:91,1] = PR[GP1:90,1] + -26.019;
   1:  PR[GP1:91,2] = PR[GP1:90,2] + 39.886;
   1:L PR[91] 10mm/sec CNT100;
   1:  PR[GP1:91,1] = PR[GP1:90,1] + -26.217;
   1:  PR[GP1:91,2] = PR[GP1:90,2] + 39.849;
   1:L PR[91] 10mm/sec CNT100;
   1:  PR[GP1:91,1] = PR[GP1:90,1] + -31.301;
   1:  PR[GP1:91,2] = PR[GP1:90,2] + 37.541;
   1:L PR[91] 10mm/sec CNT100;
   1:  PR[GP1:91,1] = PR[GP1:90,1] + -38.786;
   1:  PR[GP1:91,2] = PR[GP1:90,2] + 34.269;
   1:L PR[91] 10mm/sec CNT100;
   1:  PR[GP1:91,1] = PR[GP1:90,1] + -38.876;
   1:  PR[GP1:91,2] = PR[GP1:90,2] + 34.212;
   1:L PR[91] 10mm/sec CNT100;
   1:  PR[GP1:91,1] = PR[GP1:90,1] + -48.945;
   1:  PR[GP1:91,2] = PR[GP1:90,2] + 25.084;
   1:L PR[91] 10mm/sec CNT100;
   1:  PR[GP1:91,1] = PR[GP1:90,1] + -49.163;
   1:  PR[GP1:91,2] = PR[GP1:90,2] + 24.744;
   1:L PR[91] 10mm/sec CNT100;
   1:  PR[GP1:91,1] = PR[GP1:90,1] + -55.331;
   1:  PR[GP1:91,2] = PR[GP1:90,2] + 13.603;
   1:L PR[91] 10mm/sec CNT100;
   1:  PR[GP1:91,1] = PR[GP1:90,1] + -55.519;
   1:  PR[GP1:91,2] = PR[GP1:90,2] + 13.084;
   1:L PR[91] 10mm/sec CNT100;
   1:  PR[GP1:91,1] = PR[GP1:90,1] + -55.586;
   1:  PR[GP1:91,2] = PR[GP1:90,2] + 12.484;
   1:L PR[91] 10mm/sec CNT100;
   1:  PR[GP1:91,1] = PR[GP1:90,1] + -57.678;
   1:  PR[GP1:91,2] = PR[GP1:90,2] + 0.261;
   1:L PR[91] 10mm/sec CNT100;
   1:  PR[GP1:91,1] = PR[GP1:90,1] + -57.610;
   1:  PR[GP1:91,2] = PR[GP1:90,2] + -0.345;
   1:L PR[91] 10mm/sec CNT100;
   1:  PR[GP1:91,1] = PR[GP1:90,1] + -55.534;
   1:  PR[GP1:91,2] = PR[GP1:90,2] + -12.484;
   1:L PR[91] 10mm/sec CNT100;
   1:  PR[GP1:91,1] = PR[GP1:90,1] + -55.340;
   1:  PR[GP1:91,2] = PR[GP1:90,2] + -13.021;
   1:L PR[91] 10mm/sec CNT100;
   1:  PR[GP1:91,1] = PR[GP1:90,1] + -49.198;
   1:  PR[GP1:91,2] = PR[GP1:90,2] + -24.142;
   1:L PR[91] 10mm/sec CNT100;
   1:  PR[GP1:91,1] = PR[GP1:90,1] + -48.974;
   1:  PR[GP1:91,2] = PR[GP1:90,2] + -24.492;
   1:L PR[91] 10mm/sec CNT100;
   1:  PR[GP1:91,1] = PR[GP1:90,1] + -48.700;
   1:  PR[GP1:91,2] = PR[GP1:90,2] + -24.761;
   1:L PR[91] 10mm/sec CNT100;
   1:  PR[GP1:91,1] = PR[GP1:90,1] + -38.951;
   1:  PR[GP1:91,2] = PR[GP1:90,2] + -33.605;
   1:L PR[91] 10mm/sec CNT100;
   1:  PR[GP1:91,1] = PR[GP1:90,1] + -38.858;
   1:  PR[GP1:91,2] = PR[GP1:90,2] + -33.663;
   1:L PR[91] 10mm/sec CNT100;
   1:  PR[GP1:91,1] = PR[GP1:90,1] + -31.302;
   1:  PR[GP1:91,2] = PR[GP1:90,2] + -36.989;
   1:L PR[91] 10mm/sec CNT100;
   1:  PR[GP1:91,1] = PR[GP1:90,1] + -26.331;
   1:  PR[GP1:91,2] = PR[GP1:90,2] + -39.260;
   1:L PR[91] 10mm/sec CNT100;
   1:  PR[GP1:91,1] = PR[GP1:90,1] + -26.138;
   1:  PR[GP1:91,2] = PR[GP1:90,2] + -39.296;
   1:L PR[91] 10mm/sec CNT100;
   1:  PR[GP1:91,1] = PR[GP1:90,1] + -12.552;
   1:  PR[GP1:91,2] = PR[GP1:90,2] + -40.787;
   1:L PR[91] 10mm/sec CNT100;
   1:  PR[GP1:91,1] = PR[GP1:90,1] + -11.675;
   1:  PR[GP1:91,2] = PR[GP1:90,2] + -40.640;
   1:L PR[91] 10mm/sec CNT100;
   1:  PR[GP1:91,1] = PR[GP1:90,1] + -0.263;
   1:  PR[GP1:91,2] = PR[GP1:90,2] + -38.186;
   1:L PR[91] 10mm/sec CNT100;
   1:  PR[GP1:91,1] = PR[GP1:90,1] + 10.712;
   1:  PR[GP1:91,2] = PR[GP1:90,2] + -40.727;
   1:  PR[GP1:91,3] = PR[GP1:90,3] + 89.365;
   1:L PR[91] 10mm/sec CNT100;
   1:  PR[GP1:91,1] = PR[GP1:90,1] + 11.836;
   1:  PR[GP1:91,2] = PR[GP1:90,2] + -40.916;
   1:L PR[91] 10mm/sec CNT100;
   1:  PR[GP1:91,1] = PR[GP1:90,1] + 25.211;
   1:  PR[GP1:91,2] = PR[GP1:90,2] + -39.446;
   1:L PR[91] 10mm/sec CNT100;
   1:  PR[GP1:91,1] = PR[GP1:90,1] + 25.678;
   1:  PR[GP1:91,2] = PR[GP1:90,2] + -39.359;
   1:L PR[91] 10mm/sec CNT100;
   1:  PR[GP1:91,1] = PR[GP1:90,1] + 35.459;
   1:  PR[GP1:91,2] = PR[GP1:90,2] + -34.894;
   1:L PR[91] 10mm/sec CNT100;
   1:  PR[GP1:91,1] = PR[GP1:90,1] + 38.175;
   1:  PR[GP1:91,2] = PR[GP1:90,2] + -33.700;
   1:L PR[91] 10mm/sec CNT100;
   1:  PR[GP1:91,1] = PR[GP1:90,1] + 48.263;
   1:  PR[GP1:91,2] = PR[GP1:90,2] + -24.520;
   1:L PR[91] 10mm/sec CNT100;
   1:  PR[GP1:91,1] = PR[GP1:90,1] + 48.409;
   1:  PR[GP1:91,2] = PR[GP1:90,2] + -24.294;
   1:L PR[91] 10mm/sec CNT100;
   1:  PR[GP1:91,1] = PR[GP1:90,1] + 54.658;
   1:  PR[GP1:91,2] = PR[GP1:90,2] + -12.999;
   1:L PR[91] 10mm/sec CNT100;
   1:  PR[GP1:91,1] = PR[GP1:90,1] + 54.800;
   1:  PR[GP1:91,2] = PR[GP1:90,2] + -12.613;
   1:L PR[91] 10mm/sec CNT100;
   1:  PR[GP1:91,1] = PR[GP1:90,1] + 54.854;
   1:  PR[GP1:91,2] = PR[GP1:90,2] + -12.133;
   1:L PR[91] 10mm/sec CNT100;
   1:  PR[GP1:91,1] = PR[GP1:90,1] + 56.974;
   1:  PR[GP1:91,2] = PR[GP1:90,2] + 0.296;
   1:L PR[91] 10mm/sec CNT100;
   1:  PR[GP1:91,1] = PR[GP1:90,1] + 56.919;
   1:  PR[GP1:91,2] = PR[GP1:90,2] + 0.787;
   1:L PR[91] 10mm/sec CNT100;
   1:  PR[GP1:91,1] = PR[GP1:90,1] + 54.797;
   1:  PR[GP1:91,2] = PR[GP1:90,2] + 13.181;
   1:L PR[91] 10mm/sec CNT100;
   1:  PR[GP1:91,1] = PR[GP1:90,1] + 54.649;
   1:  PR[GP1:91,2] = PR[GP1:90,2] + 13.582;
   1:L PR[91] 10mm/sec CNT100;
   1:  PR[GP1:91,1] = PR[GP1:90,1] + 48.374;
   1:  PR[GP1:91,2] = PR[GP1:90,2] + 24.897;
   1:L PR[91] 10mm/sec CNT100;
   1:  PR[GP1:91,1] = PR[GP1:90,1] + 48.222;
   1:  PR[GP1:91,2] = PR[GP1:90,2] + 25.132;
   1:L PR[91] 10mm/sec CNT100;
   1:  PR[GP1:91,1] = PR[GP1:90,1] + 48.039;
   1:  PR[GP1:91,2] = PR[GP1:90,2] + 25.312;
   1:L PR[91] 10mm/sec CNT100;
   1:  PR[GP1:91,1] = PR[GP1:90,1] + 38.101;
   1:  PR[GP1:91,2] = PR[GP1:90,2] + 34.306;
   1:L PR[91] 10mm/sec CNT100;
   1:  PR[GP1:91,1] = PR[GP1:90,1] + 35.460;
   1:  PR[GP1:91,2] = PR[GP1:90,2] + 35.460;
   1:L PR[91] 10mm/sec CNT100;
   1:  PR[GP1:91,1] = PR[GP1:90,1] + 25.567;
   1:  PR[GP1:91,2] = PR[GP1:90,2] + 39.948;
   1:L PR[91] 10mm/sec CNT100;
   1:  PR[GP1:91,1] = PR[GP1:90,1] + 25.094;
   1:  PR[GP1:91,2] = PR[GP1:90,2] + 40.036;
   1:L PR[91] 10mm/sec CNT100;
   1:  PR[GP1:91,1] = PR[GP1:90,1] + 11.700;
   1:  PR[GP1:91,2] = PR[GP1:90,2] + 41.466;
   1:L PR[91] 10mm/sec CNT100;
   1:  PR[GP1:91,1] = PR[GP1:90,1] + 10.085;
   1:  PR[GP1:91,2] = PR[GP1:90,2] + 41.182;
   1:L PR[91] 10mm/sec CNT100;
   1:  PR[GP1:91,1] = PR[GP1:90,1] + -0.260;
   1:  PR[GP1:91,2] = PR[GP1:90,2] + 38.926;
   1:L PR[91] 10mm/sec CNT100;
   1:  PR[GP1:91,1] = PR[GP1:90,1] + -10.610;
   1:  PR[GP1:91,2] = PR[GP1:90,2] + 41.182;
   1:L PR[91] 10mm/sec CNT100;
   1:  PR[GP1:91,1] = PR[GP1:90,1] + -12.226;
   1:  PR[GP1:91,2] = PR[GP1:90,2] + 41.466;
   1:L PR[91] 10mm/sec CNT100;
   1:  PR[GP1:91,1] = PR[GP1:90,1] + -25.620;
   1:  PR[GP1:91,2] = PR[GP1:90,2] + 40.037;
   1:L PR[91] 10mm/sec CNT100;
   1:  PR[GP1:91,1] = PR[GP1:90,1] + -26.093;
   1:  PR[GP1:91,2] = PR[GP1:90,2] + 39.949;
   1:L PR[91] 10mm/sec CNT100;
   1:  PR[GP1:91,1] = PR[GP1:90,1] + -35.986;
   1:  PR[GP1:91,2] = PR[GP1:90,2] + 35.458;
   1:L PR[91] 10mm/sec CNT100;
   1:  PR[GP1:91,1] = PR[GP1:90,1] + -38.627;
   1:  PR[GP1:91,2] = PR[GP1:90,2] + 34.303;
   1:L PR[91] 10mm/sec CNT100;
   1:  PR[GP1:91,1] = PR[GP1:90,1] + -48.757;
   1:  PR[GP1:91,2] = PR[GP1:90,2] + 25.127;
   1:L PR[91] 10mm/sec CNT100;
   1:  PR[GP1:91,1] = PR[GP1:90,1] + -48.900;
   1:  PR[GP1:91,2] = PR[GP1:90,2] + 24.904;
   1:L PR[91] 10mm/sec CNT100;
   1:  PR[GP1:91,1] = PR[GP1:90,1] + -55.176;
   1:  PR[GP1:91,2] = PR[GP1:90,2] + 13.568;
   1:L PR[91] 10mm/sec CNT100;
   1:  PR[GP1:91,1] = PR[GP1:90,1] + -55.319;
   1:  PR[GP1:91,2] = PR[GP1:90,2] + 13.174;
   1:L PR[91] 10mm/sec CNT100;
   1:  PR[GP1:91,1] = PR[GP1:90,1] + -55.372;
   1:  PR[GP1:91,2] = PR[GP1:90,2] + 12.704;
   1:L PR[91] 10mm/sec CNT100;
   1:  PR[GP1:91,1] = PR[GP1:90,1] + -57.501;
   1:  PR[GP1:91,2] = PR[GP1:90,2] + 0.261;
   1:L PR[91] 10mm/sec CNT100;
   1:  PR[GP1:91,1] = PR[GP1:90,1] + -57.447;
   1:  PR[GP1:91,2] = PR[GP1:90,2] + -0.217;
   1:L PR[91] 10mm/sec CNT100;
   1:  PR[GP1:91,1] = PR[GP1:90,1] + -55.334;
   1:  PR[GP1:91,2] = PR[GP1:90,2] + -12.574;
   1:L PR[91] 10mm/sec CNT100;
   1:  PR[GP1:91,1] = PR[GP1:90,1] + -55.185;
   1:  PR[GP1:91,2] = PR[GP1:90,2] + -12.984;
   1:L PR[91] 10mm/sec CNT100;
   1:  PR[GP1:91,1] = PR[GP1:90,1] + -48.936;
   1:  PR[GP1:91,2] = PR[GP1:90,2] + -24.300;
   1:L PR[91] 10mm/sec CNT100;
   1:  PR[GP1:91,1] = PR[GP1:90,1] + -48.786;
   1:  PR[GP1:91,2] = PR[GP1:90,2] + -24.535;
   1:L PR[91] 10mm/sec CNT100;
   1:  PR[GP1:91,1] = PR[GP1:90,1] + -48.602;
   1:  PR[GP1:91,2] = PR[GP1:90,2] + -24.715;
   1:L PR[91] 10mm/sec CNT100;
   1:  PR[GP1:91,1] = PR[GP1:90,1] + -38.702;
   1:  PR[GP1:91,2] = PR[GP1:90,2] + -33.697;
   1:L PR[91] 10mm/sec CNT100;
   1:  PR[GP1:91,1] = PR[GP1:90,1] + -35.987;
   1:  PR[GP1:91,2] = PR[GP1:90,2] + -34.892;
   1:L PR[91] 10mm/sec CNT100;
   1:  PR[GP1:91,1] = PR[GP1:90,1] + -26.204;
   1:  PR[GP1:91,2] = PR[GP1:90,2] + -39.360;
   1:L PR[91] 10mm/sec CNT100;
   1:  PR[GP1:91,1] = PR[GP1:90,1] + -25.738;
   1:  PR[GP1:91,2] = PR[GP1:90,2] + -39.448;
   1:L PR[91] 10mm/sec CNT100;
   1:  PR[GP1:91,1] = PR[GP1:90,1] + -12.363;
   1:  PR[GP1:91,2] = PR[GP1:90,2] + -40.915;
   1:L PR[91] 10mm/sec CNT100;
   1:  PR[GP1:91,1] = PR[GP1:90,1] + -11.237;
   1:  PR[GP1:91,2] = PR[GP1:90,2] + -40.727;
   1:L PR[91] 10mm/sec CNT100;
   1:  PR[GP1:91,1] = PR[GP1:90,1] + -0.263;
   1:  PR[GP1:91,2] = PR[GP1:90,2] + -38.367;
   1:L PR[91] 10mm/sec CNT100;
   1:  PR[GP1:91,1] = PR[GP1:90,1] + 10.274;
   1:  PR[GP1:91,2] = PR[GP1:90,2] + -40.814;
   1:  PR[GP1:91,3] = PR[GP1:90,3] + 89.975;
   1:L PR[91] 10mm/sec CNT100;
   1:  PR[GP1:91,1] = PR[GP1:90,1] + 11.647;
   1:  PR[GP1:91,2] = PR[GP1:90,2] + -41.044;
   1:L PR[91] 10mm/sec CNT100;
   1:  PR[GP1:91,1] = PR[GP1:90,1] + 24.811;
   1:  PR[GP1:91,2] = PR[GP1:90,2] + -39.598;
   1:L PR[91] 10mm/sec CNT100;
   1:  PR[GP1:91,1] = PR[GP1:90,1] + 25.552;
   1:  PR[GP1:91,2] = PR[GP1:90,2] + -39.460;
   1:L PR[91] 10mm/sec CNT100;
   1:  PR[GP1:91,1] = PR[GP1:90,1] + 37.963;
   1:  PR[GP1:91,2] = PR[GP1:90,2] + -33.794;
   1:L PR[91] 10mm/sec CNT100;
   1:  PR[GP1:91,1] = PR[GP1:90,1] + 37.986;
   1:  PR[GP1:91,2] = PR[GP1:90,2] + -33.780;
   1:L PR[91] 10mm/sec CNT100;
   1:  PR[GP1:91,1] = PR[GP1:90,1] + 39.988;
   1:  PR[GP1:91,2] = PR[GP1:90,2] + -31.919;
   1:L PR[91] 10mm/sec CNT100;
   1:  PR[GP1:91,1] = PR[GP1:90,1] + 48.076;
   1:  PR[GP1:91,2] = PR[GP1:90,2] + -24.562;
   1:L PR[91] 10mm/sec CNT100;
   1:  PR[GP1:91,1] = PR[GP1:90,1] + 48.148;
   1:  PR[GP1:91,2] = PR[GP1:90,2] + -24.451;
   1:L PR[91] 10mm/sec CNT100;
   1:  PR[GP1:91,1] = PR[GP1:90,1] + 54.504;
   1:  PR[GP1:91,2] = PR[GP1:90,2] + -12.962;
   1:L PR[91] 10mm/sec CNT100;
   1:  PR[GP1:91,1] = PR[GP1:90,1] + 54.600;
   1:  PR[GP1:91,2] = PR[GP1:90,2] + -12.700;
   1:L PR[91] 10mm/sec CNT100;
   1:  PR[GP1:91,1] = PR[GP1:90,1] + 54.640;
   1:  PR[GP1:91,2] = PR[GP1:90,2] + -12.353;
   1:L PR[91] 10mm/sec CNT100;
   1:  PR[GP1:91,1] = PR[GP1:90,1] + 56.797;
   1:  PR[GP1:91,2] = PR[GP1:90,2] + 0.296;
   1:L PR[91] 10mm/sec CNT100;
   1:  PR[GP1:91,1] = PR[GP1:90,1] + 56.756;
   1:  PR[GP1:91,2] = PR[GP1:90,2] + 0.656;
   1:L PR[91] 10mm/sec CNT100;
   1:  PR[GP1:91,1] = PR[GP1:90,1] + 54.597;
   1:  PR[GP1:91,2] = PR[GP1:90,2] + 13.268;
   1:L PR[91] 10mm/sec CNT100;
   1:  PR[GP1:91,1] = PR[GP1:90,1] + 54.495;
   1:  PR[GP1:91,2] = PR[GP1:90,2] + 13.546;
   1:L PR[91] 10mm/sec CNT100;
   1:  PR[GP1:91,1] = PR[GP1:90,1] + 48.111;
   1:  PR[GP1:91,2] = PR[GP1:90,2] + 25.055;
   1:L PR[91] 10mm/sec CNT100;
   1:  PR[GP1:91,1] = PR[GP1:90,1] + 48.034;
   1:  PR[GP1:91,2] = PR[GP1:90,2] + 25.175;
   1:L PR[91] 10mm/sec CNT100;
   1:  PR[GP1:91,1] = PR[GP1:90,1] + 47.941;
   1:  PR[GP1:91,2] = PR[GP1:90,2] + 25.266;
   1:L PR[91] 10mm/sec CNT100;
   1:  PR[GP1:91,1] = PR[GP1:90,1] + 39.989;
   1:  PR[GP1:91,2] = PR[GP1:90,2] + 32.463;
   1:L PR[91] 10mm/sec CNT100;
   1:  PR[GP1:91,1] = PR[GP1:90,1] + 37.913;
   1:  PR[GP1:91,2] = PR[GP1:90,2] + 34.386;
   1:L PR[91] 10mm/sec CNT100;
   1:  PR[GP1:91,1] = PR[GP1:90,1] + 37.886;
   1:  PR[GP1:91,2] = PR[GP1:90,2] + 34.403;
   1:L PR[91] 10mm/sec CNT100;
   1:  PR[GP1:91,1] = PR[GP1:90,1] + 25.443;
   1:  PR[GP1:91,2] = PR[GP1:90,2] + 40.047;
   1:L PR[91] 10mm/sec CNT100;
   1:  PR[GP1:91,1] = PR[GP1:90,1] + 24.695;
   1:  PR[GP1:91,2] = PR[GP1:90,2] + 40.187;
   1:L PR[91] 10mm/sec CNT100;
   1:  PR[GP1:91,1] = PR[GP1:90,1] + 11.513;
   1:  PR[GP1:91,2] = PR[GP1:90,2] + 41.595;
   1:L PR[91] 10mm/sec CNT100;
   1:  PR[GP1:91,1] = PR[GP1:90,1] + 9.552;
   1:  PR[GP1:91,2] = PR[GP1:90,2] + 41.250;
   1:L PR[91] 10mm/sec CNT100;
   1:  PR[GP1:91,1] = PR[GP1:90,1] + -0.260;
   1:  PR[GP1:91,2] = PR[GP1:90,2] + 39.110;
   1:L PR[91] 10mm/sec CNT100;
   1:  PR[GP1:91,1] = PR[GP1:90,1] + -10.076;
   1:  PR[GP1:91,2] = PR[GP1:90,2] + 41.250;
   1:L PR[91] 10mm/sec CNT100;
   1:  PR[GP1:91,1] = PR[GP1:90,1] + -12.039;
   1:  PR[GP1:91,2] = PR[GP1:90,2] + 41.594;
   1:L PR[91] 10mm/sec CNT100;
   1:  PR[GP1:91,1] = PR[GP1:90,1] + -25.222;
   1:  PR[GP1:91,2] = PR[GP1:90,2] + 40.188;
   1:L PR[91] 10mm/sec CNT100;
   1:  PR[GP1:91,1] = PR[GP1:90,1] + -25.968;
   1:  PR[GP1:91,2] = PR[GP1:90,2] + 40.049;
   1:L PR[91] 10mm/sec CNT100;
   1:  PR[GP1:91,1] = PR[GP1:90,1] + -38.412;
   1:  PR[GP1:91,2] = PR[GP1:90,2] + 34.400;
   1:L PR[91] 10mm/sec CNT100;
   1:  PR[GP1:91,1] = PR[GP1:90,1] + -38.440;
   1:  PR[GP1:91,2] = PR[GP1:90,2] + 34.383;
   1:L PR[91] 10mm/sec CNT100;
   1:  PR[GP1:91,1] = PR[GP1:90,1] + -40.515;
   1:  PR[GP1:91,2] = PR[GP1:90,2] + 32.462;
   1:L PR[91] 10mm/sec CNT100;
   1:  PR[GP1:91,1] = PR[GP1:90,1] + -48.568;
   1:  PR[GP1:91,2] = PR[GP1:90,2] + 25.171;
   1:L PR[91] 10mm/sec CNT100;
   1:  PR[GP1:91,1] = PR[GP1:90,1] + -48.638;
   1:  PR[GP1:91,2] = PR[GP1:90,2] + 25.063;
   1:L PR[91] 10mm/sec CNT100;
   1:  PR[GP1:91,1] = PR[GP1:90,1] + -55.021;
   1:  PR[GP1:91,2] = PR[GP1:90,2] + 13.532;
   1:L PR[91] 10mm/sec CNT100;
   1:  PR[GP1:91,1] = PR[GP1:90,1] + -55.119;
   1:  PR[GP1:91,2] = PR[GP1:90,2] + 13.264;
   1:L PR[91] 10mm/sec CNT100;
   1:  PR[GP1:91,1] = PR[GP1:90,1] + -55.157;
   1:  PR[GP1:91,2] = PR[GP1:90,2] + 12.924;
   1:L PR[91] 10mm/sec CNT100;
   1:  PR[GP1:91,1] = PR[GP1:90,1] + -57.324;
   1:  PR[GP1:91,2] = PR[GP1:90,2] + 0.261;
   1:L PR[91] 10mm/sec CNT100;
   1:  PR[GP1:91,1] = PR[GP1:90,1] + -57.285;
   1:  PR[GP1:91,2] = PR[GP1:90,2] + -0.089;
   1:L PR[91] 10mm/sec CNT100;
   1:  PR[GP1:91,1] = PR[GP1:90,1] + -55.134;
   1:  PR[GP1:91,2] = PR[GP1:90,2] + -12.663;
   1:L PR[91] 10mm/sec CNT100;
   1:  PR[GP1:91,1] = PR[GP1:90,1] + -55.031;
   1:  PR[GP1:91,2] = PR[GP1:90,2] + -12.948;
   1:L PR[91] 10mm/sec CNT100;
   1:  PR[GP1:91,1] = PR[GP1:90,1] + -48.674;
   1:  PR[GP1:91,2] = PR[GP1:90,2] + -24.458;
   1:L PR[91] 10mm/sec CNT100;
   1:  PR[GP1:91,1] = PR[GP1:90,1] + -48.598;
   1:  PR[GP1:91,2] = PR[GP1:90,2] + -24.578;
   1:L PR[91] 10mm/sec CNT100;
   1:  PR[GP1:91,1] = PR[GP1:90,1] + -48.504;
   1:  PR[GP1:91,2] = PR[GP1:90,2] + -24.669;
   1:L PR[91] 10mm/sec CNT100;
   1:  PR[GP1:91,1] = PR[GP1:90,1] + -40.516;
   1:  PR[GP1:91,2] = PR[GP1:90,2] + -31.916;
   1:L PR[91] 10mm/sec CNT100;
   1:  PR[GP1:91,1] = PR[GP1:90,1] + -38.513;
   1:  PR[GP1:91,2] = PR[GP1:90,2] + -33.776;
   1:L PR[91] 10mm/sec CNT100;
   1:  PR[GP1:91,1] = PR[GP1:90,1] + -38.489;
   1:  PR[GP1:91,2] = PR[GP1:90,2] + -33.791;
   1:L PR[91] 10mm/sec CNT100;
   1:  PR[GP1:91,1] = PR[GP1:90,1] + -26.078;
   1:  PR[GP1:91,2] = PR[GP1:90,2] + -39.461;
   1:L PR[91] 10mm/sec CNT100;
   1:  PR[GP1:91,1] = PR[GP1:90,1] + -25.337;
   1:  PR[GP1:91,2] = PR[GP1:90,2] + -39.599;
   1:L PR[91] 10mm/sec CNT100;
   1:  PR[GP1:91,1] = PR[GP1:90,1] + -12.174;
   1:  PR[GP1:91,2] = PR[GP1:90,2] + -41.044;
   1:L PR[91] 10mm/sec CNT100;
   1:  PR[GP1:91,1] = PR[GP1:90,1] + -10.799;
   1:  PR[GP1:91,2] = PR[GP1:90,2] + -40.813;
   1:L PR[91] 10mm/sec CNT100;
   1:  PR[GP1:91,1] = PR[GP1:90,1] + -0.262;
   1:  PR[GP1:91,2] = PR[GP1:90,2] + -38.548;
   1:L PR[91] 10mm/sec CNT100;
   1:  PR[GP1:91,1] = PR[GP1:90,1] + 9.836;
   1:  PR[GP1:91,2] = PR[GP1:90,2] + -40.900;
   1:  PR[GP1:91,3] = PR[GP1:90,3] + 90.585;
   1:L PR[91] 10mm/sec CNT100;
   1:  PR[GP1:91,1] = PR[GP1:90,1] + 11.458;
   1:  PR[GP1:91,2] = PR[GP1:90,2] + -41.173;
   1:L PR[91] 10mm/sec CNT100;
   1:  PR[GP1:91,1] = PR[GP1:90,1] + 24.410;
   1:  PR[GP1:91,2] = PR[GP1:90,2] + -39.750;
   1:L PR[91] 10mm/sec CNT100;
   1:  PR[GP1:91,1] = PR[GP1:90,1] + 25.425;
   1:  PR[GP1:91,2] = PR[GP1:90,2] + -39.560;
   1:L PR[91] 10mm/sec CNT100;
   1:  PR[GP1:91,1] = PR[GP1:90,1] + 37.637;
   1:  PR[GP1:91,2] = PR[GP1:90,2] + -33.985;
   1:L PR[91] 10mm/sec CNT100;
   1:  PR[GP1:91,1] = PR[GP1:90,1] + 37.908;
   1:  PR[GP1:91,2] = PR[GP1:90,2] + -33.818;
   1:L PR[91] 10mm/sec CNT100;
   1:  PR[GP1:91,1] = PR[GP1:90,1] + 44.684;
   1:  PR[GP1:91,2] = PR[GP1:90,2] + -27.519;
   1:L PR[91] 10mm/sec CNT100;
   1:  PR[GP1:91,1] = PR[GP1:90,1] + 47.874;
   1:  PR[GP1:91,2] = PR[GP1:90,2] + -24.617;
   1:L PR[91] 10mm/sec CNT100;
   1:  PR[GP1:91,1] = PR[GP1:90,1] + 54.350;
   1:  PR[GP1:91,2] = PR[GP1:90,2] + -12.925;
   1:L PR[91] 10mm/sec CNT100;
   1:  PR[GP1:91,1] = PR[GP1:90,1] + 54.401;
   1:  PR[GP1:91,2] = PR[GP1:90,2] + -12.786;
   1:L PR[91] 10mm/sec CNT100;
   1:  PR[GP1:91,1] = PR[GP1:90,1] + 54.425;
   1:  PR[GP1:91,2] = PR[GP1:90,2] + -12.573;
   1:L PR[91] 10mm/sec CNT100;
   1:  PR[GP1:91,1] = PR[GP1:90,1] + 56.620;
   1:  PR[GP1:91,2] = PR[GP1:90,2] + 0.296;
   1:L PR[91] 10mm/sec CNT100;
   1:  PR[GP1:91,1] = PR[GP1:90,1] + 56.594;
   1:  PR[GP1:91,2] = PR[GP1:90,2] + 0.525;
   1:L PR[91] 10mm/sec CNT100;
   1:  PR[GP1:91,1] = PR[GP1:90,1] + 54.397;
   1:  PR[GP1:91,2] = PR[GP1:90,2] + 13.355;
   1:L PR[91] 10mm/sec CNT100;
   1:  PR[GP1:91,1] = PR[GP1:90,1] + 54.340;
   1:  PR[GP1:91,2] = PR[GP1:90,2] + 13.509;
   1:L PR[91] 10mm/sec CNT100;
   1:  PR[GP1:91,1] = PR[GP1:90,1] + 47.865;
   1:  PR[GP1:91,2] = PR[GP1:90,2] + 25.186;
   1:L PR[91] 10mm/sec CNT100;
   1:  PR[GP1:91,1] = PR[GP1:90,1] + 47.818;
   1:  PR[GP1:91,2] = PR[GP1:90,2] + 25.243;
   1:L PR[91] 10mm/sec CNT100;
   1:  PR[GP1:91,1] = PR[GP1:90,1] + 44.685;
   1:  PR[GP1:91,2] = PR[GP1:90,2] + 28.079;
   1:L PR[91] 10mm/sec CNT100;
   1:  PR[GP1:91,1] = PR[GP1:90,1] + 37.836;
   1:  PR[GP1:91,2] = PR[GP1:90,2] + 34.423;
   1:L PR[91] 10mm/sec CNT100;
   1:  PR[GP1:91,1] = PR[GP1:90,1] + 37.562;
   1:  PR[GP1:91,2] = PR[GP1:90,2] + 34.593;
   1:L PR[91] 10mm/sec CNT100;
   1:  PR[GP1:91,1] = PR[GP1:90,1] + 25.318;
   1:  PR[GP1:91,2] = PR[GP1:90,2] + 40.147;
   1:L PR[91] 10mm/sec CNT100;
   1:  PR[GP1:91,1] = PR[GP1:90,1] + 24.297;
   1:  PR[GP1:91,2] = PR[GP1:90,2] + 40.338;
   1:L PR[91] 10mm/sec CNT100;
   1:  PR[GP1:91,1] = PR[GP1:90,1] + 11.326;
   1:  PR[GP1:91,2] = PR[GP1:90,2] + 41.723;
   1:L PR[91] 10mm/sec CNT100;
   1:  PR[GP1:91,1] = PR[GP1:90,1] + 9.019;
   1:  PR[GP1:91,2] = PR[GP1:90,2] + 41.318;
   1:L PR[91] 10mm/sec CNT100;
   1:  PR[GP1:91,1] = PR[GP1:90,1] + -0.260;
   1:  PR[GP1:91,2] = PR[GP1:90,2] + 39.294;
   1:L PR[91] 10mm/sec CNT100;
   1:  PR[GP1:91,1] = PR[GP1:90,1] + -9.542;
   1:  PR[GP1:91,2] = PR[GP1:90,2] + 41.317;
   1:L PR[91] 10mm/sec CNT100;
   1:  PR[GP1:91,1] = PR[GP1:90,1] + -11.852;
   1:  PR[GP1:91,2] = PR[GP1:90,2] + 41.723;
   1:L PR[91] 10mm/sec CNT100;
   1:  PR[GP1:91,1] = PR[GP1:90,1] + -24.823;
   1:  PR[GP1:91,2] = PR[GP1:90,2] + 40.339;
   1:L PR[91] 10mm/sec CNT100;
   1:  PR[GP1:91,1] = PR[GP1:90,1] + -25.844;
   1:  PR[GP1:91,2] = PR[GP1:90,2] + 40.149;
   1:L PR[91] 10mm/sec CNT100;
   1:  PR[GP1:91,1] = PR[GP1:90,1] + -38.088;
   1:  PR[GP1:91,2] = PR[GP1:90,2] + 34.590;
   1:L PR[91] 10mm/sec CNT100;
   1:  PR[GP1:91,1] = PR[GP1:90,1] + -38.362;
   1:  PR[GP1:91,2] = PR[GP1:90,2] + 34.420;
   1:L PR[91] 10mm/sec CNT100;
   1:  PR[GP1:91,1] = PR[GP1:90,1] + -45.212;
   1:  PR[GP1:91,2] = PR[GP1:90,2] + 28.083;
   1:L PR[91] 10mm/sec CNT100;
   1:  PR[GP1:91,1] = PR[GP1:90,1] + -48.365;
   1:  PR[GP1:91,2] = PR[GP1:90,2] + 25.228;
   1:L PR[91] 10mm/sec CNT100;
   1:  PR[GP1:91,1] = PR[GP1:90,1] + -54.867;
   1:  PR[GP1:91,2] = PR[GP1:90,2] + 13.496;
   1:L PR[91] 10mm/sec CNT100;
   1:  PR[GP1:91,1] = PR[GP1:90,1] + -54.918;
   1:  PR[GP1:91,2] = PR[GP1:90,2] + 13.354;
   1:L PR[91] 10mm/sec CNT100;
   1:  PR[GP1:91,1] = PR[GP1:90,1] + -54.942;
   1:  PR[GP1:91,2] = PR[GP1:90,2] + 13.144;
   1:L PR[91] 10mm/sec CNT100;
   1:  PR[GP1:91,1] = PR[GP1:90,1] + -57.146;
   1:  PR[GP1:91,2] = PR[GP1:90,2] + 0.261;
   1:L PR[91] 10mm/sec CNT100;
   1:  PR[GP1:91,1] = PR[GP1:90,1] + -57.122;
   1:  PR[GP1:91,2] = PR[GP1:90,2] + 0.039;
   1:L PR[91] 10mm/sec CNT100;
   1:  PR[GP1:91,1] = PR[GP1:90,1] + -54.934;
   1:  PR[GP1:91,2] = PR[GP1:90,2] + -12.752;
   1:L PR[91] 10mm/sec CNT100;
   1:  PR[GP1:91,1] = PR[GP1:90,1] + -54.876;
   1:  PR[GP1:91,2] = PR[GP1:90,2] + -12.911;
   1:L PR[91] 10mm/sec CNT100;
   1:  PR[GP1:91,1] = PR[GP1:90,1] + -48.428;
   1:  PR[GP1:91,2] = PR[GP1:90,2] + -24.588;
   1:L PR[91] 10mm/sec CNT100;
   1:  PR[GP1:91,1] = PR[GP1:90,1] + -48.380;
   1:  PR[GP1:91,2] = PR[GP1:90,2] + -24.647;
   1:L PR[91] 10mm/sec CNT100;
   1:  PR[GP1:91,1] = PR[GP1:90,1] + -45.213;
   1:  PR[GP1:91,2] = PR[GP1:90,2] + -27.521;
   1:L PR[91] 10mm/sec CNT100;
   1:  PR[GP1:91,1] = PR[GP1:90,1] + -38.434;
   1:  PR[GP1:91,2] = PR[GP1:90,2] + -33.815;
   1:L PR[91] 10mm/sec CNT100;
   1:  PR[GP1:91,1] = PR[GP1:90,1] + -38.163;
   1:  PR[GP1:91,2] = PR[GP1:90,2] + -33.983;
   1:L PR[91] 10mm/sec CNT100;
   1:  PR[GP1:91,1] = PR[GP1:90,1] + -25.952;
   1:  PR[GP1:91,2] = PR[GP1:90,2] + -39.561;
   1:L PR[91] 10mm/sec CNT100;
   1:  PR[GP1:91,1] = PR[GP1:90,1] + -24.937;
   1:  PR[GP1:91,2] = PR[GP1:90,2] + -39.751;
   1:L PR[91] 10mm/sec CNT100;
   1:  PR[GP1:91,1] = PR[GP1:90,1] + -11.985;
   1:  PR[GP1:91,2] = PR[GP1:90,2] + -41.172;
   1:L PR[91] 10mm/sec CNT100;
   1:  PR[GP1:91,1] = PR[GP1:90,1] + -10.361;
   1:  PR[GP1:91,2] = PR[GP1:90,2] + -40.900;
   1:L PR[91] 10mm/sec CNT100;
   1:  PR[GP1:91,1] = PR[GP1:90,1] + -0.262;
   1:  PR[GP1:91,2] = PR[GP1:90,2] + -38.728;
   1:L PR[91] 10mm/sec CNT100;
   1:  PR[GP1:91,1] = PR[GP1:90,1] + 9.398;
   1:  PR[GP1:91,2] = PR[GP1:90,2] + -40.987;
   1:  PR[GP1:91,3] = PR[GP1:90,3] + 91.195;
   1:L PR[91] 10mm/sec CNT100;
   1:  PR[GP1:91,1] = PR[GP1:90,1] + 11.268;
   1:  PR[GP1:91,2] = PR[GP1:90,2] + -41.301;
   1:L PR[91] 10mm/sec CNT100;
